    if(wv_seq[0] == 0 or wv_seq[0] == 3):
      if(a9_wv_weldingon==True):
        program_weld_on = False
        if(isHicomm):
          write_port_register(202,0)
          write_port_register(149,0)
        else:
          set_standard_digital_out(0,False)
        end
        if(wv_weldpar[2]==1):
          target_pos = feature_offset(get_actual_tcp_pose(),p[0,0,-0.01,0,0,0],wv_Line_Feature2)
          movel(target_pos,0.5,0.01)
        end
      end
    end
    background_pose = [dumy_p,dumy_p,dumy_p]
    move_p = background_pose
    return sin_dir
  end
  $ 150 "Reset"
  $ 151 "If Reset_Trig"
  if (Reset_Trig):
    $ 152 "Reset_Trig≔ False "
    global Reset_Trig=  False
    $ 153 "Call robotand_cell_initalizat"
    robotand_cell_initalizat()
    $ 154 "Auto_trig≔ False "
    global Auto_trig=  False
    $ 155 "write_port_register(cell_3f_2f_151,0)"
    write_port_register(cell_3f_2f_151,0)
    $ 156 "write_port_register(cell_info_152,0)"
    write_port_register(cell_info_152,0)
    $ 157 "write_port_register(weld_req_153,0)"
    write_port_register(weld_req_153,0)
    $ 158 "write_port_register(return_done_240,0)"
    write_port_register(return_done_240,0)
    $ 159 "write_port_register(robot_move_163,0)"
    write_port_register(robot_move_163,0)
    $ 160 "write_port_register(robot_pose_164,0)"
    write_port_register(robot_pose_164,0)
    $ 161 "write_port_register(182,0)"
    write_port_register(182,0)
    $ 162 "write_port_register(185,0)"
    write_port_register(185,0)
    $ 163 "write_port_register(201,0)"
    write_port_register(201,0)
    $ 164 "write_port_register(202,0)"
    write_port_register(202,0)
  end
  $ 165 "Welding_Init"
  $ 166 "'welding parameter initialization'"
  # 'welding parameter initialization'
  $ 167 "welding_etc"
  $ 195 "c5_wv_gap_y≔0"
  global c5_wv_gap_y=0
  $ 196 "c6_wv_gap_cpm≔0"
  global c6_wv_gap_cpm=0
  $ 197 "c9_wv_gap_freq≔0"
  global c9_wv_gap_freq=0
  $ 198 "c4_gap_enable≔0"
  global c4_gap_enable=0
  $ 199 "c7_wv_gap≔[c4_gap_enable,c5_wv_gap_y,c6_wv_gap_cpm,c9_wv_gap_freq]"
  global c7_wv_gap=[c4_gap_enable,c5_wv_gap_y,c6_wv_gap_cpm,c9_wv_gap_freq]
  $ 200 "init_reset_modbus_server"
  $ 201 "set_tool_voltage(24)"
  set_tool_voltage(24)
  $ 202 "write_port_register(163,0)"
  write_port_register(163,0)
  $ 203 "write_port_register(164,0)"
  write_port_register(164,0)
  $ 205 "write_port_register(201,1)"
  write_port_register(201,1)
  $ 206 "write_port_register(202,0)"
  write_port_register(202,0)
  $ 1235 "Thread_2"
  thread Thread_2():
    while (True):
      $ 1236 "heartbeat≔heartbeat+1"
      global heartbeat=heartbeat+1
      $ 1237 "If heartbeat>499"
      if (heartbeat>499):
        $ 1238 "heartbeat≔0"
        global heartbeat=0
      end
      $ 1239 "write_port_register(128,heartbeat)"
      write_port_register(128,heartbeat)
      $ 1249 "Wait: 1.0"
      sleep(1.0)
    end
  end
  threadId_Thread_2 = run Thread_2()
  $ 1250 "Thread_1"
  thread Thread_1():
    while (True):
      $ 1251 "a0_Job_Mode≔read_port_register(162)"
      global a0_Job_Mode= read_port_register (162)
      $ 1252 "a1_job_move≔read_port_register(163)"
      global a1_job_move= read_port_register (163)
      $ 1253 "If red_led≟ True "
      if (get_tool_digital_out(0) ==   True  ):
        $ 1254 "Set red_led=Off"
        set_tool_digital_out(0, False)
      end
      $ 1255 "If a0_Job_Mode≟2"
      if (a0_Job_Mode == 2):
        $ 1256 "If read_port_register(arc_onoff_168)≟2"
        if ( read_port_register (arc_onoff_168) == 2):
          $ 1257 "a9_wv_weldingon≔ True "
          global a9_wv_weldingon=  True
        else:
          $ 1258 "Else" "noBreak"
          $ 1259 "a9_wv_weldingon≔ False "
          global a9_wv_weldingon=  False
        end
        $ 1260 "If Auto_trig"
        if (Auto_trig):
          $ 1261 "get_next_number≔read_port_register(166)"
          global get_next_number= read_port_register (166)
          $ 1262 "get_move_trig≔read_port_register(167)"
          global get_move_trig= read_port_register (167)
          $ 1263 "If get_move_trig≟1 and running_trig≟ True "
          if (get_move_trig == 1  and  running_trig ==   True  ):
            $ 1264 "If get_next_number<0 or get_next_number>30"
            if (get_next_number<0  or  get_next_number>30):
              $ 1265 "write_port_register(142,141)"
              write_port_register(142,141)
              $ 1266 "Halt"
              halt
            end
            $ 1267 "If get_next_number≠Auto_cur_cell"
            if (get_next_number != Auto_cur_cell):
              $ 1268 "running_trig≔ False "
              global running_trig=  False
              $ 1269 "write_welder(0, False )"
              write_welder(0,  False  )
              $ 1270 "write_port_register(149,0)"
              write_port_register(149,0)
              $ 1271 "write_port_register(202,0)"
              write_port_register(202,0)
            else:
              $ 1272 "Else" "noBreak"
              $ 1273 "write_port_register(166,0)"
              write_port_register(166,0)
              $ 1274 "write_port_register(167,0)"
              write_port_register(167,0)
            end
          end
        end
        $ 1275 "If t_time>timer_1"
        if (t_time>timer_1):
          $ 1276 "write_port_register(143,timer_1)"
          write_port_register(143,timer_1)
        else:
          $ 1277 "Else" "noBreak"
          $ 1278 "write_port_register(143,timer_1)"
          write_port_register(143,timer_1)
          $ 1279 "write_port_register(144,timer_1)"
          write_port_register(144,timer_1)
        end
        $ 1280 "Monitoring touch and welding"
        $ 1281 "If read_welder_control(0) and read_port_register(130)≠1"
        if (read_welder_control(0)  and   read_port_register (130) != 1):
          $ 1282 "write_port_register(130,1)"
          write_port_register(130,1)
        else:
          $ 1283 "ElseIf read_welder_control(0) and read_port_register(130)≠0"
          if (read_welder_control(0)  and   read_port_register (130) != 0):
            $ 1284 "write_port_register(130,0)"
            write_port_register(130,0)
          end
        end
        $ 1285 "If read_welder(5)"
        if (read_welder(5)):
          $ 1286 "'check wcr in (digital)'"
          # 'check wcr in (digital)'
          $ 1287 "write_output_float_register(20,1)"
          write_output_float_register(20,1)
        else:
          $ 1288 "Else" "noBreak"
          $ 1289 "write_output_float_register(20,0)"
          write_output_float_register(20,0)
        end
        $ 1290 "If read_welder(4)"
        if (read_welder(4)):
          $ 1291 "'check touch (digital)'"
          # 'check touch (digital)'
          $ 1292 "write_output_float_register(21,1)"
          write_output_float_register(21,1)
        else:
          $ 1293 "Else" "noBreak"
          $ 1294 "write_output_float_register(21,0)"
          write_output_float_register(21,0)
        end
        $ 1295 "If read_welder_control(0)"
        if (read_welder_control(0)):
          $ 1296 "'check welding out (digital)'"
          # 'check welding out (digital)'
          $ 1297 "write_output_float_register(17,1)"
          write_output_float_register(17,1)
        else:
          $ 1298 "Else" "noBreak"
          $ 1299 "write_output_float_register(17,0)"
          write_output_float_register(17,0)
        end
        $ 1300 "If read_welder_control(4)"
        if (read_welder_control(4)):
          $ 1301 "'check touch out (digital)'"
          # 'check touch out (digital)'
          $ 1302 "write_output_float_register(18,1)"
          write_output_float_register(18,1)
        else:
          $ 1303 "Else" "noBreak"
          $ 1304 "write_output_float_register(18,0)"
          write_output_float_register(18,0)
        end
      end
      $ 1305 "If get_tool_digital_in(1)≟ True "
      if (get_tool_digital_in(1) ==   True  ):
        $ 1306 "set_tool_digital_out(1, False )"
        set_tool_digital_out(1,  False  )
      else:
        $ 1307 "Else" "noBreak"
        $ 1308 "set_tool_digital_out(1, True )"
        set_tool_digital_out(1,  True  )
      end
      $ 1309 "If red_led≟ True "
      if (get_tool_digital_out(0) ==   True  ):
        $ 1310 "Set red_led=Off"
        set_tool_digital_out(0, False)
        $ 1311 "end_freedrive_mode()"
        end_freedrive_mode()
      end
      $ 1312 "check_speed()"
      check_speed()
      $ 1313 "Wait: 0.05"
      sleep(0.05)
    end
  end
  threadId_Thread_1 = run Thread_1()
  thread EventThread():
    while (True):
      if (event_cal_on):
        $ 1317 "move_i_f≔1"
        global move_i_f=1
        $ 1318 "get_pose_side≔0"
        global get_pose_side=0
        $ 1319 "Loop move_i_f<10"
        while (move_i_f<10):
          $ 1320 "If A_Touch_trig_l[move_i_f]≟ True "
          if (A_Touch_trig_l[move_i_f] ==   True  ):
            $ 1321 "If move_i_f≟A_VL1 or move_i_f≟A_VL2"
            if (move_i_f == A_VL1  or  move_i_f == A_VL2):
              $ 1322 "A_sel_v≔move_i_f"
              global A_sel_v=move_i_f
              $ 1323 "If simulation_mode"
              if (simulation_mode):
                $ 1324 "Call welding_parameter_sim"
                welding_parameter_sim()
              else:
                $ 1325 "Else" "noBreak"
                $ 1326 "Call welding_parameter_init"
                welding_parameter_init()
              end
              $ 1327 "If a8_wv_distance<5"
              if (a8_wv_distance<5):
                $ 1328 "write_port_register(142,143)"
                write_port_register(142,143)
                $ 1329 "Halt"
                halt
              end
              $ 1330 "b2_left_par≔ True "
              global b2_left_par=  True
              $ 1331 "b8_wv_2f≔ False "
              global b8_wv_2f=  False
              $ 1332 "If move_i_f≟A_VL2"
              if (move_i_f == A_VL2):
                $ 1333 "callar_hor≔a6_callar_hor"
                global callar_hor=a6_callar_hor
                $ 1334 "b2_cell≔0"
                global b2_cell=0
                $ 1335 "If b1_cell_info_L≟c or b1_cell_info_L≟d"
                if (b1_cell_info_L == c  or  b1_cell_info_L == d):
                  $ 1336 "b2_cell≔b1_cell_info_L"
                  global b2_cell=b1_cell_info_L
                else:
                  $ 1337 "Else" "noBreak"
                  $ 1338 "b2_cell≔0"
                  global b2_cell=0
                end
              else:
                $ 1339 "Else" "noBreak"
                $ 1340 "callar_hor≔0"
                global callar_hor=0
                $ 1341 "b2_cell≔b1_cell_info_L"
                global b2_cell=b1_cell_info_L
              end
              $ 1342 "get_pos≔get_lr(left,a6_f_width,a5_f_hole,a7_f_distance,b2_left_par,b8_wv_2f,Touch_dis,get_margin_z,get_pose_side,callar_hor,b2_cell,center_line)"
              global get_pos=get_lr(p[.480496318984, .411279115151, .006998291210, -2.211681476386, -.899147924387, -1.383032568605],a6_f_width,a5_f_hole,a7_f_distance,b2_left_par,b8_wv_2f,Touch_dis,get_margin_z,get_pose_side,callar_hor,b2_cell,center_line)
              $ 1343 "pre_tp≔tilt_3f_fun(get_pos,[0,0,0],0)"
              global pre_tp=tilt_3f_fun(get_pos,[0,0,0],0)
              $ 1344 "A_Prepos_l[move_i_f]=pre_tp"
              A_Prepos_l[move_i_f]=pre_tp
            else:
              $ 1345 "ElseIf move_i_f≟A_VR1 or move_i_f≟A_VR2"
              if (move_i_f == A_VR1  or  move_i_f == A_VR2):
                $ 1346 "A_sel_v≔move_i_f"
                global A_sel_v=move_i_f
                $ 1347 "If simulation_mode"
                if (simulation_mode):
                  $ 1348 "Call welding_parameter_sim"
                  welding_parameter_sim()
                else:
                  $ 1349 "Else" "noBreak"
                  $ 1350 "Call welding_parameter_init"
                  welding_parameter_init()
                end
                $ 1351 "If a8_wv_distance<5"
                if (a8_wv_distance<5):
                  $ 1352 "write_port_register(142,143)"
                  write_port_register(142,143)
                  $ 1353 "Halt"
                  halt
                end
                $ 1354 "b2_left_par≔ False "
                global b2_left_par=  False
                $ 1355 "b8_wv_2f≔ False "
                global b8_wv_2f=  False
                $ 1356 "If move_i_f≟A_VR2"
                if (move_i_f == A_VR2):
                  $ 1357 "callar_hor≔a6_callar_hor"
                  global callar_hor=a6_callar_hor
                  $ 1358 "If b1_cell_info_R≟c or b1_cell_info_R≟d"
                  if (b1_cell_info_R == c  or  b1_cell_info_R == d):
                    $ 1359 "b2_cell≔b1_cell_info_R"
                    global b2_cell=b1_cell_info_R
                  else:
                    $ 1360 "Else" "noBreak"
                    $ 1361 "b2_cell≔0"
                    global b2_cell=0
                  end
                else:
                  $ 1362 "Else" "noBreak"
                  $ 1363 "callar_hor≔0"
                  global callar_hor=0
                  $ 1364 "b2_cell≔b1_cell_info_R"
                  global b2_cell=b1_cell_info_R
                end
                $ 1365 "get_pos≔get_lr(right,a6_f_width,a5_f_hole,a7_f_distance,b2_left_par,b8_wv_2f,Touch_dis,get_margin_z,get_pose_side,callar_hor,b2_cell,center_line)"
                global get_pos=get_lr(p[.475000000000, -.421403215678, .026417194146, 1.917761036827, -1.141682393512, 1.523356199292],a6_f_width,a5_f_hole,a7_f_distance,b2_left_par,b8_wv_2f,Touch_dis,get_margin_z,get_pose_side,callar_hor,b2_cell,center_line)
                $ 1366 "pre_tp≔tilt_3f_fun(get_pos,[0,0,0],0)"
                global pre_tp=tilt_3f_fun(get_pos,[0,0,0],0)
                $ 1367 "A_Prepos_l[move_i_f]=pre_tp"
                A_Prepos_l[move_i_f]=pre_tp
              else:
                $ 1368 "ElseIf move_i_f≟A_HOR"
                if (move_i_f == A_HOR):
                  $ 1369 "A_sel_v≔A_HOR"
                  global A_sel_v=A_HOR
                  $ 1370 "If simulation_mode"
                  if (simulation_mode):
                    $ 1371 "Call welding_parameter_sim"
                    welding_parameter_sim()
                  else:
                    $ 1372 "Else" "noBreak"
                    $ 1373 "Call welding_parameter_init"
                    welding_parameter_init()
                  end
                  $ 1374 "b8_wv_2f≔ True "
                  global b8_wv_2f=  True
                  $ 1375 "b2_left_par≔ True "
                  global b2_left_par=  True
                  $ 1376 "b2_cell≔b1_cell_info_L"
                  global b2_cell=b1_cell_info_L
                  $ 1377 "get_pos≔get_lr(up_left,a6_f_width,a5_f_hole,a7_f_distance,b2_left_par,b8_wv_2f,Touch_dis,get_margin_z,get_pose_side,0,b2_cell,center_line)"
                  global get_pos=get_lr(p[.492775857339, .409517380626, -.029063830209, -2.419264859926, -.998084331190, -1.368689080860],a6_f_width,a5_f_hole,a7_f_distance,b2_left_par,b8_wv_2f,Touch_dis,get_margin_z,get_pose_side,0,b2_cell,center_line)
                  $ 1378 "pre_tp≔get_pos"
                  global pre_tp=get_pos
                  $ 1379 "A_Prepos_l[move_i_f]=pre_tp"
                  A_Prepos_l[move_i_f]=pre_tp
                else:
                  $ 1380 "ElseIf move_i_f≟A_HOR_R"
                  if (move_i_f == A_HOR_R):
                    $ 1381 "A_sel_v≔A_HOR"
                    global A_sel_v=A_HOR
                    $ 1382 "If simulation_mode"
                    if (simulation_mode):
                      $ 1383 "Call welding_parameter_sim"
                      welding_parameter_sim()
                    else:
                      $ 1384 "Else" "noBreak"
                      $ 1385 "Call welding_parameter_init"
                      welding_parameter_init()
                    end
                    $ 1386 "b2_left_par≔ False "
                    global b2_left_par=  False
                    $ 1387 "b8_wv_2f≔ True "
                    global b8_wv_2f=  True
                    $ 1388 "b2_cell≔b1_cell_info_R"
                    global b2_cell=b1_cell_info_R
                    $ 1389 "get_pos≔get_lr(up_right,a6_f_width,a5_f_hole,a7_f_distance,b2_left_par,b8_wv_2f,Touch_dis,get_margin_z,get_pose_side,0,b2_cell,center_line)"
                    global get_pos=get_lr(p[.445203173045, -.406687378356, -.031125942276, 2.308490741423, -1.066468937023, 1.322151316133],a6_f_width,a5_f_hole,a7_f_distance,b2_left_par,b8_wv_2f,Touch_dis,get_margin_z,get_pose_side,0,b2_cell,center_line)
                    $ 1390 "pre_tp≔get_pos"
                    global pre_tp=get_pos
                    $ 1391 "A_Prepos_l[move_i_f]=pre_tp"
                    A_Prepos_l[move_i_f]=pre_tp
                  else:
                    $ 1392 "ElseIf move_i_f≟A_HOR_ML"
                    if (move_i_f == A_HOR_ML):
                      $ 1393 "A_sel_v≔A_HOR_ML"
                      global A_sel_v=A_HOR_ML
                      $ 1394 "If simulation_mode"
                      if (simulation_mode):
                        $ 1395 "Call welding_parameter_sim"
                        welding_parameter_sim()
                      else:
                        $ 1396 "Else" "noBreak"
                        $ 1397 "Call welding_parameter_init"
                        welding_parameter_init()
                      end
                      $ 1398 "b8_wv_2f≔ True "
                      global b8_wv_2f=  True
                      $ 1399 "b2_left_par≔ True "
                      global b2_left_par=  True
                      $ 1400 "b2_cell≔b1_cell_info_L"
                      global b2_cell=b1_cell_info_L
                      $ 1401 "Touch_dis≔-1*Touch_dis"
                      global Touch_dis=-1*Touch_dis
                      $ 1402 "get_pos≔get_lr(up_left,a6_f_width,a5_f_hole,a7_f_distance,b2_left_par,b8_wv_2f,Touch_dis,get_margin_z,get_pose_side,a6_callar_hor,b2_cell,center_line)"
                      global get_pos=get_lr(p[.492775857339, .409517380626, -.029063830209, -2.419264859926, -.998084331190, -1.368689080860],a6_f_width,a5_f_hole,a7_f_distance,b2_left_par,b8_wv_2f,Touch_dis,get_margin_z,get_pose_side,a6_callar_hor,b2_cell,center_line)
                      $ 1403 "Touch_dis≔-1*Touch_dis"
                      global Touch_dis=-1*Touch_dis
                      $ 1404 "pre_tp≔get_pos"
                      global pre_tp=get_pos
                      $ 1405 "A_Prepos_l[move_i_f]=pre_tp"
                      A_Prepos_l[move_i_f]=pre_tp
                    else:
                      $ 1406 "ElseIf move_i_f≟A_HOR_MR"
                      if (move_i_f == A_HOR_MR):
                        $ 1407 "A_sel_v≔A_HOR_MR"
                        global A_sel_v=A_HOR_MR
                        $ 1408 "If simulation_mode"
                        if (simulation_mode):
                          $ 1409 "Call welding_parameter_sim"
                          welding_parameter_sim()
                        else:
                          $ 1410 "Else" "noBreak"
                          $ 1411 "Call welding_parameter_init"
                          welding_parameter_init()
                        end
                        $ 1412 "b2_left_par≔ False "
                        global b2_left_par=  False
                        $ 1413 "b8_wv_2f≔ True "
                        global b8_wv_2f=  True
                        $ 1414 "b2_cell≔b1_cell_info_R"
                        global b2_cell=b1_cell_info_R
                        $ 1415 "Touch_dis≔-1*Touch_dis"
                        global Touch_dis=-1*Touch_dis
                        $ 1416 "get_pos≔get_lr(up_right,a6_f_width,a5_f_hole,a7_f_distance,b2_left_par,b8_wv_2f,Touch_dis,get_margin_z,get_pose_side,a6_callar_hor,b2_cell,center_line)"
                        global get_pos=get_lr(p[.445203173045, -.406687378356, -.031125942276, 2.308490741423, -1.066468937023, 1.322151316133],a6_f_width,a5_f_hole,a7_f_distance,b2_left_par,b8_wv_2f,Touch_dis,get_margin_z,get_pose_side,a6_callar_hor,b2_cell,center_line)
                        $ 1417 "Touch_dis≔-1*Touch_dis"
                        global Touch_dis=-1*Touch_dis
                        $ 1418 "pre_tp≔get_pos"
                        global pre_tp=get_pos
                        $ 1419 "A_Prepos_l[move_i_f]=pre_tp"
                        A_Prepos_l[move_i_f]=pre_tp
                      end
                    end
                  end
                end
              end
            end
            $ 1420 "If move_i_f≤4"
            if (move_i_f <= 4):
              $ 1421 "A_Prepos_l[move_i_f+9]=p[0,0,0,0,0,0]"
              A_Prepos_l[move_i_f+9]=p[0,0,0,0,0,0]
            end
          end
          $ 1424 "move_i_f≔move_i_f+1"
          global move_i_f=move_i_f+1
        end
        $ 1425 "event_cal_on≔ False "
        global event_cal_on=  False
      elif (event_side_on):
        $ 1429 "Wait event_cal_on≟ False "
        while (not(event_cal_on ==   False  )):
          sync()
        end
        $ 1430 "move_i_f≔1"
        global move_i_f=1
        $ 1431 "get_pose_side≔get_pose_side_t"
        global get_pose_side=get_pose_side_t
        $ 1432 "Loop move_i_f<10"
        while (move_i_f<10):
          $ 1433 "If A_Touch_trig_l[move_i_f]≟ True "
          if (A_Touch_trig_l[move_i_f] ==   True  ):
            $ 1434 "If move_i_f≟A_VL1 or move_i_f≟A_VL2"
            if (move_i_f == A_VL1  or  move_i_f == A_VL2):
              $ 1435 "A_Prepos_l[move_i_f]=side_apply(A_Prepos_l[move_i_f],center_line,get_pose_side)"
              A_Prepos_l[move_i_f]=side_apply(A_Prepos_l[move_i_f],center_line,get_pose_side)
            else:
              $ 1436 "ElseIf move_i_f≟A_VR1 or move_i_f≟A_VR2"
              if (move_i_f == A_VR1  or  move_i_f == A_VR2):
                $ 1437 "A_Prepos_l[move_i_f]=side_apply(A_Prepos_l[move_i_f],center_line,get_pose_side)"
                A_Prepos_l[move_i_f]=side_apply(A_Prepos_l[move_i_f],center_line,get_pose_side)
              else:
                $ 1438 "ElseIf move_i_f≟A_HOR"
                if (move_i_f == A_HOR):
                  $ 1439 "A_Prepos_l[move_i_f]=side_apply(A_Prepos_l[move_i_f],center_line,get_pose_side)"
                  A_Prepos_l[move_i_f]=side_apply(A_Prepos_l[move_i_f],center_line,get_pose_side)
                else:
                  $ 1440 "ElseIf move_i_f≟A_HOR_R"
                  if (move_i_f == A_HOR_R):
                    $ 1441 "A_Prepos_l[move_i_f]=side_apply(A_Prepos_l[move_i_f],center_line,get_pose_side)"
                    A_Prepos_l[move_i_f]=side_apply(A_Prepos_l[move_i_f],center_line,get_pose_side)
                  else:
                    $ 1442 "ElseIf move_i_f≟A_HOR_ML"
                    if (move_i_f == A_HOR_ML):
                      $ 1443 "A_Prepos_l[move_i_f]=side_apply(A_Prepos_l[move_i_f],center_line,get_pose_side)"
                      A_Prepos_l[move_i_f]=side_apply(A_Prepos_l[move_i_f],center_line,get_pose_side)
                    else:
                      $ 1444 "ElseIf move_i_f≟A_HOR_MR"
                      if (move_i_f == A_HOR_MR):
                        $ 1445 "A_Prepos_l[move_i_f]=side_apply(A_Prepos_l[move_i_f],center_line,get_pose_side)"
                        A_Prepos_l[move_i_f]=side_apply(A_Prepos_l[move_i_f],center_line,get_pose_side)
                      end
                    end
                  end
                end
              end
            end
          end
          $ 1446 "move_i_f≔move_i_f+1"
          global move_i_f=move_i_f+1
        end
        $ 1447 "event_side_on≔ False "
        global event_side_on=  False
      elif (reset_trig):
        $ 1449 "Call reset_weld_param"
        reset_weld_param()
        $ 1450 "reset_trig≔ False "
        global reset_trig=  False
      elif (time_cal_trig):
        $ 1452 "t_time≔time_cal(Auto_W_num,Auto_total_cell,A_Speed_list,A_Distance_list,A_Touch_p,0)"
        global t_time=time_cal(Auto_W_num,Auto_total_cell,A_Speed_list,A_Distance_list,A_Touch_p,0)
        $ 1453 "write_port_register(144,t_time)"
        write_port_register(144,t_time)
        $ 1454 "time_cal_trig≔ False "
        global time_cal_trig=  False
      elif (pause_trig):
        $ 1456 "s_conn≔socket_open('192.168.1.7',29999)"
        global s_conn=socket_open("192.168.1.7",29999)
        $ 1457 "s_send≔socket_send_string('pause')"
        global s_send=socket_send_string("pause")
        $ 1458 "s_send≔socket_send_byte(10)"
        global s_send=socket_send_byte(10)
        $ 1459 "socket_close()"
        socket_close()
        $ 1460 "pause_trig≔ False "
        global pause_trig=  False
      end
      sync()
    end
  end
  eventThread = run EventThread()
  while (True):
    $ 207 "Robot Program"
    $ 225 "If simulation_mode"
    if (simulation_mode):
      $ 226 "'work mode 2'"
      # 'work mode 2'
      $ 227 "write_port_register(162,2)"
      write_port_register(162,2)
      $ 228 "touch_temp≔0"
      global touch_temp=0
    end
    $ 229 "If a0_Job_Mode≟1"
    if (a0_Job_Mode == 1):
      $ 230 "job mode 1"
      $ 231 "'JOB_MANUAL'"
      # 'JOB_MANUAL'
      $ 232 "write_port_register(robot_ready_141,1)"
      write_port_register(robot_ready_141,1)
      $ 233 "If freedrive≟ True  and freedrive_trg≟ False "
      if (get_tool_digital_in(1) ==   True    and  freedrive_trg ==   False  ):
        $ 234 "freedrive_trg≔ True "
        global freedrive_trg=  True
        $ 235 "freedrive_mode()"
        freedrive_mode()
      else:
        $ 236 "ElseIf freedrive≟ False  and freedrive_trg≟ True "
        if (get_tool_digital_in(1) ==   False    and  freedrive_trg ==   True  ):
          $ 237 "end_freedrive_mode()"
          end_freedrive_mode()
          $ 238 "freedrive_trg≔ False "
          global freedrive_trg=  False
        end
      end
      $ 242 "If freedrive≟ True  and save_tool≟ True "
      if (get_tool_digital_in(1) ==   True    and  get_tool_digital_in(0) ==   True  ):
        $ 246 "Wait: 0.01"
        sleep(0.01)
      else:
        $ 247 "ElseIf a1_job_move≟1"
        if (a1_job_move == 1):
          $ 248 "'Manual - Move Home/Packing/Warmup'"
          # 'Manual - Move Home/Packing/Warmup'
          $ 249 "If read_port_register(robot_pose_164)≟1"
          if ( read_port_register (robot_pose_164) == 1):
            $ 250 "write_port_register(robot_ready_141,0)"
            write_port_register(robot_ready_141,0)
            $ 251 "homeing()"
            homeing()
            $ 252 "MoveJ"
            $ 253 "Packing_pos" "breakAfter"
            movej([1.5877798795700073, -0.0173419157611292, -2.4983108679400843, -1.4065726439105433, 1.626846194267273, 3.0169763565063477], a=0.9599310885968813, v=0.9599310885968813)
          else:
            $ 254 "ElseIf read_port_register(robot_pose_164)≟2"
            if ( read_port_register (robot_pose_164) == 2):
              $ 255 "write_port_register(robot_ready_141,0)"
              write_port_register(robot_ready_141,0)
              $ 256 "homeing()"
              homeing()
            else:
              $ 257 "ElseIf read_port_register(robot_pose_164)≟3"
              global thread_flag_257=0
              thread Thread_if_257():
                $ 258 "write_port_register(robot_ready_141,0)"
                write_port_register(robot_ready_141,0)
                $ 259 "Warm-up"
                $ 260 "Loop 22 times"
                Loop_9 = 0
                while (Loop_9 < 22):
                  $ 261 "MoveJ"
                  $ 262 "Warming_1" "breakAfter"
                  movej([1.3388409470167426, -1.0894445773085817, -1.21578769245379, -2.340308120379028, 1.4975742894997062, 2.3546781160711117], a=0.5235987755982988, v=0.2617993877991494)
                  $ 263 "Warming_2" "breakAfter"
                  movej([0.3765170846483107, -1.0894466320678031, -1.215768207322279, -2.3402268007341895, 1.4977834941028334, 2.3545507363355367], a=0.5235987755982988, v=0.2617993877991494)
                  $ 264 "Warming_3" "breakAfter"
                  movej([0.70229908534082, -1.0894474234917375, -1.2158576930717002, -2.340314378048955, 1.497725846219038, 2.3545705560997385], a=0.5235987755982988, v=0.2617993877991494)
                  $ 265 "Warming_4" "breakAfter"
                  movej([0.7262700130956564, -1.3120291852612347, -1.2099656497338014, -2.3525900953229293, 1.4887798341942113, 2.3787312683819053], a=0.5235987755982988, v=0.2617993877991494)
                  $ 266 "Wariming_5" "breakAfter"
                  movej([0.6926726182060315, -1.0476106481659855, -1.2179788018883642, -2.3355421428203886, 1.501172277634622, 2.3452576869092923], a=0.5235987755982988, v=0.2617993877991494)
                  $ 267 "Warming_6" "breakAfter"
                  movej([0.706544616734295, -1.047040496424307, -1.4190888321133315, -2.3436933501169452, 1.4896422361111494, 2.359727124413684], a=0.5235987755982988, v=0.2617993877991494)
                  $ 268 "Warming_7" "breakAfter"
                  movej([0.6929880468286825, -1.0476354157293724, -1.2203987593812862, -2.335678707355349, 1.5010671072282735, 2.34550338764565], a=0.5235987755982988, v=0.2617993877991494)
                  $ 269 "Warming_8" "breakAfter"
                  movej([0.6920775233962951, -1.0506328608604214, -1.2152130579572011, -2.5072867131215766, 1.4917910996963177, 2.3459413556024855], a=0.5235987755982988, v=0.2617993877991494)
                  $ 270 "Warming_9" "breakAfter"
                  movej([0.692933302781529, -1.0474869681006531, -1.2206503884398048, -2.327559666709858, 1.5015191668476027, 2.3454614641680087], a=0.5235987755982988, v=0.2617993877991494)
                  $ 271 "Warming_10" "breakAfter"
                  movej([0.7189566793816887, -1.1462083943843844, -1.3286482352122917, -2.3898368690561114, 1.223390234561962, 2.3705741030878644], a=0.5235987755982988, v=0.2617993877991494)
                  $ 272 "Warming_11" "breakAfter"
                  movej([0.6952417412291937, -1.0226626805382075, -1.3187663864026051, -2.3852732107244847, 1.5281305955128988, 2.3484138521676003], a=0.5235987755982988, v=0.2617993877991494)
                  $ 273 "Warming_12" "breakAfter"
                  movej([0.6939658935868351, -1.0222541193887693, -1.3205060700309819, -2.4036431483224994, 1.8876292979334401, 2.3447872177861786], a=0.5235987755982988, v=0.2617993877991494)
                  $ 274 "Warming_13" "breakAfter"
                  movej([0.6855475262233561, -1.0389108716421376, -1.3163550590643318, -2.371185255756596, 1.5282046997566647, 1.6427118007650936], a=0.5235987755982988, v=0.2617993877991494)
                  $ 275 "Warming_14" "breakAfter"
                  movej([0.721349856763205, -1.0075982028648234, -1.3205933019427434, -2.399656340024448, 1.5281938267886401, 2.9170078642332813], a=0.5235987755982988, v=0.2617993877991494)
                  Loop_9 = Loop_9 + 1
                end
                $ 276 "homeing()"
                homeing()
                $ 277 "Wait: 2.0"
                sleep(2.0)
                thread_flag_257 = 1
              end
              if ( read_port_register (robot_pose_164) == 3):
                global thread_handler_257=run Thread_if_257()
                while (thread_flag_257 == 0):
                  if not( read_port_register (robot_pose_164) == 3):
                    kill thread_handler_257
                    thread_flag_257 = 2
                  else:
                    sync()
                  end
                end
              else:
                thread_flag_257 = 2
              end
              if (thread_flag_257 == 2):
                $ 278 "ElseIf read_port_register(robot_pose_164)≟4"
                if ( read_port_register (robot_pose_164) == 4):
                  $ 279 "write_port_register(robot_ready_141,0)"
                  write_port_register(robot_ready_141,0)
                  $ 280 "homeing()"
                  homeing()
                  $ 281 "MoveJ"
                  $ 282 "pre_mounting" "breakAfter"
                  movej([1.2356762886047363, -0.8703244368182581, -0.942230526600973, -2.3905327955829065, 1.3216267824172974, 2.6514604091644287], a=0.7853981633974483, v=0.7853981633974483)
                  $ 283 "Mounting_pos" "breakAfter"
                  movej([0.6231353085164267, -0.6300961531972575, -0.9034285948871803, -1.770059340221131, 1.417516049558281, 1.7792033261567348], a=0.7853981633974483, v=0.7853981633974483)
                else:
                  $ 284 "ElseIf read_port_register(robot_pose_164)≟5"
                  if ( read_port_register (robot_pose_164) == 5):
                    $ 285 "c_p≔get_actual_tcp_pose()"
                    global c_p= get_actual_tcp_pose ()
                    $ 286 "MoveL"
                    $ 287 "m_p≔pose_trans(c_p, p[0,0,0,d2r(tilt_deg_man),0,0])"
                    global m_p= pose_trans (c_p, p[0,0,0,d2r(tilt_deg_man),0,0])
                    $ 288 "m_p" "breakAfter"
                    movel(pose_trans(Base, m_p), a=0.03, v=0.03)
                    $ 289 "m_p≔pose_trans(c_p, p[0,0,0,d2r(-tilt_deg_man),0,0])"
                    global m_p= pose_trans (c_p, p[0,0,0,d2r(-tilt_deg_man),0,0])
                    $ 290 "m_p" "breakAfter"
                    movel(pose_trans(Base, m_p), a=0.03, v=0.03)
                    $ 291 "c_p" "breakAfter"
                    movel(pose_trans(Base, c_p), a=0.03, v=0.03)
                    $ 292 "m_p≔pose_trans(c_p, p[0,0,0,0,d2r(tilt_deg_man),0])"
                    global m_p= pose_trans (c_p, p[0,0,0,0,d2r(tilt_deg_man),0])
                    $ 293 "m_p" "breakAfter"
                    movel(pose_trans(Base, m_p), a=0.03, v=0.03)
                    $ 294 "m_p≔pose_trans(c_p, p[0,0,0,0,d2r(-tilt_deg_man),0])"
                    global m_p= pose_trans (c_p, p[0,0,0,0,d2r(-tilt_deg_man),0])
                    $ 295 "m_p" "breakAfter"
                    movel(pose_trans(Base, m_p), a=0.03, v=0.03)
                    $ 296 "c_p" "breakAfter"
                    movel(pose_trans(Base, c_p), a=0.03, v=0.03)
                    $ 297 "m_p≔pose_trans(c_p, p[0,0,0,0,0,d2r(tilt_deg_man)])"
                    global m_p= pose_trans (c_p, p[0,0,0,0,0,d2r(tilt_deg_man)])
                    $ 298 "m_p" "breakAfter"
                    movel(pose_trans(Base, m_p), a=0.03, v=0.03)
                    $ 299 "m_p≔pose_trans(c_p, p[0,0,0,0,0,d2r(-tilt_deg_man)])"
                    global m_p= pose_trans (c_p, p[0,0,0,0,0,d2r(-tilt_deg_man)])
                    $ 300 "m_p" "breakAfter"
                    movel(pose_trans(Base, m_p), a=0.03, v=0.03)
                    $ 301 "c_p" "breakAfter"
                    movel(pose_trans(Base, c_p), a=0.03, v=0.03)
                  end
                end
              end
            end
          end
          $ 302 "Call Move_done"
          Move_done()
        end
      end
      $ 303 "Call robotand_cell_initalizat"
      robotand_cell_initalizat()
    else:
      $ 304 "ElseIf a0_Job_Mode≟2"
      global thread_flag_304=0
      thread Thread_if_304():
        $ 305 "'JOB_AUTO'"
        # 'JOB_AUTO'
        $ 306 "auto_on≔ True "
        global auto_on=  True
        $ 307 "Init"
        $ 308 "If freedrive_trg"
        if (freedrive_trg):
          $ 309 "end_freedrive_mode()"
          end_freedrive_mode()
          $ 310 "freedrive_trg≔ False "
          global freedrive_trg=  False
        end
        $ 311 "write_port_register(202,0)"
        write_port_register(202,0)
        $ 312 "write_port_register(robot_ready_141,0)"
        write_port_register(robot_ready_141,0)
        $ 313 "homeing()"
        homeing()
        $ 314 "Wait: 0.2"
        sleep(0.2)
        $ 315 "Cell_calculation"
        $ 316 "'setting'"
        # 'setting'
        $ 317 "Auto_trig≔ False "
        global Auto_trig=  False
        $ 318 "If Auto_trig≟ False "
        if (Auto_trig ==   False  ):
          $ 319 "If simulation_mode"
          if (simulation_mode):
            $ 320 "b1_cell_info_L≔B"
            global b1_cell_info_L=B
            $ 321 "b1_cell_info_R≔B"
            global b1_cell_info_R=B
            $ 322 "b1_cell_select≔motion_num([A_VL1,A_VR1,A_HOR,0,0,0])"
            global b1_cell_select=motion_num([A_VL1,A_VR1,A_HOR,0,0,0])
            $ 323 "b1_cell_select≔motion_num([A_HOR,0,0,0,0,0])"
            global b1_cell_select=motion_num([A_HOR,0,0,0,0,0])
            $ 324 "EXT_flag1≔integer_to_binary_list(read_port_register(2048))"
            global EXT_flag1= integer_to_binary_list ( read_port_register (2048))
            $ 325 "b1_cell_thickne≔6"
            global b1_cell_thickne=6
            $ 326 "A_Touch_trig_l≔touch_cal(b1_cell_info_L,b1_cell_info_R,b1_cell_select)"
            global A_Touch_trig_l=touch_cal(b1_cell_info_L,b1_cell_info_R,b1_cell_select)
            $ 327 "Auto_W_num≔cell_motion(A_Touch_trig_l,b1_cell_thickne,EXT_flag1,b1_cell_info_L,b1_cell_info_R)"
            global Auto_W_num=cell_motion(A_Touch_trig_l,b1_cell_thickne,EXT_flag1,b1_cell_info_L,b1_cell_info_R)
            $ 329 "Auto_total_cell≔cell_num(Auto_W_num)"
            global Auto_total_cell=cell_num(Auto_W_num)
            $ 330 "Auto_trig≔ True "
            global Auto_trig=  True
            $ 331 "A_sel_v≔Auto_W_num[0]"
            global A_sel_v=Auto_W_num[0]
          else:
            $ 332 "Else" "noBreak"
            $ 333 "b1_cell_info_L≔read_port_register(171)"
            global b1_cell_info_L= read_port_register (171)
            $ 334 "b1_cell_info_R≔read_port_register(172)"
            global b1_cell_info_R= read_port_register (172)
            $ 335 "EXT_flag1≔integer_to_binary_list(read_port_register(179))"
            global EXT_flag1= integer_to_binary_list ( read_port_register (179))
            $ 336 "b1_cell_select≔read_port_register(178)"
            global b1_cell_select= read_port_register (178)
            $ 337 "b1_cell_thickne≔read_port_register(183)"
            global b1_cell_thickne= read_port_register (183)
            $ 338 "A_Touch_trig_l≔touch_cal(b1_cell_info_L,b1_cell_info_R,b1_cell_select)"
            global A_Touch_trig_l=touch_cal(b1_cell_info_L,b1_cell_info_R,b1_cell_select)
            $ 339 "Auto_W_num≔cell_motion(A_Touch_trig_l,b1_cell_thickne,EXT_flag1,b1_cell_info_L,b1_cell_info_R)"
            global Auto_W_num=cell_motion(A_Touch_trig_l,b1_cell_thickne,EXT_flag1,b1_cell_info_L,b1_cell_info_R)
            $ 340 "Auto_total_cell≔cell_num(Auto_W_num)"
            global Auto_total_cell=cell_num(Auto_W_num)
            $ 341 "Auto_trig≔ True "
            global Auto_trig=  True
            $ 342 "A_sel_v≔Auto_W_num[0]"
            global A_sel_v=Auto_W_num[0]
          end
          $ 343 "write_port_register(139,Auto_total_cell-1)"
          write_port_register(139,Auto_total_cell-1)
        end
        $ 344 "Auto_cur_cell≔0"
        global Auto_cur_cell=0
        $ 345 "Touch,Welding"
        $ 346 "'Calculate total sequence and decide way'"
        # 'Calculate total sequence and decide way'
        $ 347 "Calculate & Move & Touch"
        $ 348 "touch_init"
        $ 349 "Call cell_info"
        cell_info()
        $ 350 "If simulation_mode"
        if (simulation_mode):
          $ 351 "Call welding_parameter_sim"
          welding_parameter_sim()
        else:
          $ 352 "Else" "noBreak"
          $ 353 "Call welding_parameter_init"
          welding_parameter_init()
          $ 354 "touch_temp≔read_port_register(180)"
          global touch_temp= read_port_register (180)
          $ 355 "A_cur_2f≔0"
          global A_cur_2f=0
          $ 356 "wv_direction≔1"
          global wv_direction=1
        end
        $ 357 "If touch_temp≟0"
        if (touch_temp == 0):
          $ 358 "reset Variable"
          $ 359 "A_Prepos_l=[p[0, 0, 0, 0, 0, 0], p[0, 0, 0, 0, 0, 0], p[0, 0, 0, 0, 0, 0],p[0, 0, 0, 0, 0, 0], p[0, 0, 0, 0, 0, 0], p[0, 0, 0, 0, 0, 0], p[0, 0, 0, 0, 0, 0], p[0, 0, 0, 0, 0, 0], p[0, 0, 0, 0, 0, 0], p[0, 0, 0, 0, 0, 0], p[0, 0, 0, 0, 0, 0],p[0, 0, 0, 0, 0, 0],p[0, 0, 0, 0, 0, 0],p[0, 0, 0, 0, 0, 0],p[0, 0, 0, 0, 0, 0],p[0,0,0,0,0,0]]"
          A_Prepos_l=[p[0, 0, 0, 0, 0, 0], p[0, 0, 0, 0, 0, 0], p[0, 0, 0, 0, 0, 0],p[0, 0, 0, 0, 0, 0], p[0, 0, 0, 0, 0, 0], p[0, 0, 0, 0, 0, 0], p[0, 0, 0, 0, 0, 0], p[0, 0, 0, 0, 0, 0], p[0, 0, 0, 0, 0, 0], p[0, 0, 0, 0, 0, 0], p[0, 0, 0, 0, 0, 0],p[0, 0, 0, 0, 0, 0],p[0, 0, 0, 0, 0, 0],p[0, 0, 0, 0, 0, 0],p[0, 0, 0, 0, 0, 0],p[0,0,0,0,0,0]]
          $ 360 "A_Touch_p=[p[0, 0, 0, 0, 0, 0], p[0, 0, 0, 0, 0, 0], p[0, 0, 0, 0, 0, 0],p[0, 0, 0, 0, 0, 0], p[0, 0, 0, 0, 0, 0], p[0, 0, 0, 0, 0, 0], p[0, 0, 0, 0, 0, 0], p[0, 0, 0, 0, 0, 0], p[0, 0, 0, 0, 0, 0], p[0, 0, 0, 0, 0, 0], p[0, 0, 0, 0, 0, 0],p[0, 0, 0, 0, 0, 0],p[0, 0, 0, 0, 0, 0],p[0, 0, 0, 0, 0, 0],p[0, 0, 0, 0, 0, 0],p[0,0,0,0,0,0]]"
          A_Touch_p=[p[0, 0, 0, 0, 0, 0], p[0, 0, 0, 0, 0, 0], p[0, 0, 0, 0, 0, 0],p[0, 0, 0, 0, 0, 0], p[0, 0, 0, 0, 0, 0], p[0, 0, 0, 0, 0, 0], p[0, 0, 0, 0, 0, 0], p[0, 0, 0, 0, 0, 0], p[0, 0, 0, 0, 0, 0], p[0, 0, 0, 0, 0, 0], p[0, 0, 0, 0, 0, 0],p[0, 0, 0, 0, 0, 0],p[0, 0, 0, 0, 0, 0],p[0, 0, 0, 0, 0, 0],p[0, 0, 0, 0, 0, 0],p[0,0,0,0,0,0]]
          $ 361 "reset_par"
          $ 362 "for_cal_rot≔p[0,0,0,0,0,0]"
          global for_cal_rot=p[0,0,0,0,0,0]
          $ 363 "for_cal_zr≔p[0,0,0,0,0,0]"
          global for_cal_zr=p[0,0,0,0,0,0]
          $ 364 "for_cal_zl≔p[0,0,0,0,0,0]"
          global for_cal_zl=p[0,0,0,0,0,0]
          $ 365 "for_cal_x_wel≔p[0,0,0,0,0,0]"
          global for_cal_x_wel=p[0,0,0,0,0,0]
          $ 366 "for_cal_xy≔p[0,0,0,0,0,0]"
          global for_cal_xy=p[0,0,0,0,0,0]
          $ 367 "for_cal_y_wel≔p[0,0,0,0,0,0]"
          global for_cal_y_wel=p[0,0,0,0,0,0]
          $ 368 "for_x_HOR≔p[0,0,0,0,0,0]"
          global for_x_HOR=p[0,0,0,0,0,0]
          $ 369 "for_x_HOR_R≔p[0,0,0,0,0,0]"
          global for_x_HOR_R=p[0,0,0,0,0,0]
          $ 370 "for_z_VL1≔p[0,0,0,0,0,0]"
          global for_z_VL1=p[0,0,0,0,0,0]
          $ 371 "for_z_VR1≔p[0,0,0,0,0,0]"
          global for_z_VR1=p[0,0,0,0,0,0]
        end
        $ 372 "write_port_register(143,0)"
        write_port_register(143,0)
        $ 373 "write_port_register(144,0)"
        write_port_register(144,0)
        $ 374 "timer_1: Reset"
        timer_1 = 0
        $ 375 "EXT_flag1≔integer_to_binary_list(read_port_register(179))"
        global EXT_flag1= integer_to_binary_list ( read_port_register (179))
        $ 377 "If touch_temp≟0"
        if (touch_temp == 0):
          $ 378 "write_port_register(138,0)"
          write_port_register(138,0)
          $ 379 "get_touch_position"
          $ 380 "get pre-positions"
          $ 381 "If read_port_register(work_type_165)≟2"
          if ( read_port_register (work_type_165) == 2):
            $ 382 "freedrive touch"
            $ 383 "move_i≔1"
            global move_i=1
            $ 384 "Loop move_i<9"
            while (move_i<9):
              $ 385 "Wait: 0.1"
              sleep(0.1)
              $ 386 "Wait save_tool=LO"
              while (get_tool_digital_in(0) == True):
                sync()
              end
              $ 387 "If A_Touch_trig_l[move_i]≟ True "
              if (A_Touch_trig_l[move_i] ==   True  ):
                $ 388 "If move_i≟A_HOR"
                if (move_i == A_HOR):
                  $ 389 "If b1_cell_info_L≟B or b1_cell_info_L≟D or b1_cell_info_L≟d or A_Prepos_l[A_VL1]≟p[0,0,0,0,0,0]"
                  if (b1_cell_info_L == B  or  b1_cell_info_L == D  or  b1_cell_info_L == d  or  A_Prepos_l[A_VL1] == p[0,0,0,0,0,0]):
                    $ 390 "write_port_register(touch_cell_155,5)"
                    write_port_register(touch_cell_155,5)
                    $ 391 "write_port_register(touch_num_156,1)"
                    write_port_register(touch_num_156,1)
                    $ 392 "Call touch_sub"
                    touch_sub()
                    $ 393 "g_cp≔get_actual_tcp_pose()"
                    global g_cp= get_actual_tcp_pose ()
                    $ 394 "If g_cp[2]<(get_margin_z+a7_cell_bottom)/1000"
                    if (g_cp[2]<(get_margin_z+a7_cell_bottom)/1000):
                      $ 395 "g_cp[2]=(get_margin_z+a7_cell_bottom)/1000"
                      g_cp[2]=(get_margin_z+a7_cell_bottom)/1000
                    end
                    $ 396 "A_Prepos_l[move_i]=g_cp"
                    A_Prepos_l[move_i]=g_cp
                  end
                else:
                  $ 397 "ElseIf move_i≟A_HOR_ML"
                  if (move_i == A_HOR_ML):
                    $ 398 "If b1_cell_info_L≟B or b1_cell_info_L≟D or b1_cell_info_L≟d or A_Prepos_l[A_VL1]≟p[0,0,0,0,0,0]"
                    if (b1_cell_info_L == B  or  b1_cell_info_L == D  or  b1_cell_info_L == d  or  A_Prepos_l[A_VL1] == p[0,0,0,0,0,0]):
                      $ 399 "write_port_register(touch_cell_155,5)"
                      write_port_register(touch_cell_155,5)
                      $ 400 "write_port_register(touch_num_156,3)"
                      write_port_register(touch_num_156,3)
                      $ 401 "Call touch_sub"
                      touch_sub()
                      $ 402 "g_cp≔get_actual_tcp_pose()"
                      global g_cp= get_actual_tcp_pose ()
                      $ 403 "If g_cp[2]<(get_margin_z+a7_cell_bottom)/1000"
                      if (g_cp[2]<(get_margin_z+a7_cell_bottom)/1000):
                        $ 404 "g_cp[2]=(get_margin_z+a7_cell_bottom)/1000"
                        g_cp[2]=(get_margin_z+a7_cell_bottom)/1000
                      end
                      $ 405 "A_Prepos_l[move_i]=g_cp"
                      A_Prepos_l[move_i]=g_cp
                    end
                  else:
                    $ 406 "ElseIf move_i≟A_HOR_R"
                    if (move_i == A_HOR_R):
                      $ 407 "If b1_cell_info_L≟B or b1_cell_info_L≟D or b1_cell_info_L≟d or A_Prepos_l[A_VL1]≟p[0,0,0,0,0,0]"
                      if (b1_cell_info_L == B  or  b1_cell_info_L == D  or  b1_cell_info_L == d  or  A_Prepos_l[A_VL1] == p[0,0,0,0,0,0]):
                        $ 408 "write_port_register(touch_cell_155,5)"
                        write_port_register(touch_cell_155,5)
                        $ 409 "write_port_register(touch_num_156,2)"
                        write_port_register(touch_num_156,2)
                        $ 410 "Call touch_sub"
                        touch_sub()
                        $ 411 "g_cp≔get_actual_tcp_pose()"
                        global g_cp= get_actual_tcp_pose ()
                        $ 412 "If g_cp[2]<(get_margin_z+a7_cell_bottom)/1000"
                        if (g_cp[2]<(get_margin_z+a7_cell_bottom)/1000):
                          $ 413 "g_cp[2]=(get_margin_z+a7_cell_bottom)/1000"
                          g_cp[2]=(get_margin_z+a7_cell_bottom)/1000
                        end
                        $ 414 "A_Prepos_l[move_i]=g_cp"
                        A_Prepos_l[move_i]=g_cp
                      end
                    else:
                      $ 415 "ElseIf move_i≟A_HOR_MR"
                      if (move_i == A_HOR_MR):
                        $ 416 "If b1_cell_info_L≟B or b1_cell_info_L≟D or b1_cell_info_L≟d or A_Prepos_l[A_VL1]≟p[0,0,0,0,0,0]"
                        if (b1_cell_info_L == B  or  b1_cell_info_L == D  or  b1_cell_info_L == d  or  A_Prepos_l[A_VL1] == p[0,0,0,0,0,0]):
                          $ 417 "write_port_register(touch_cell_155,5)"
                          write_port_register(touch_cell_155,5)
                          $ 418 "write_port_register(touch_num_156,4)"
                          write_port_register(touch_num_156,4)
                          $ 419 "Call touch_sub"
                          touch_sub()
                          $ 420 "g_cp≔get_actual_tcp_pose()"
                          global g_cp= get_actual_tcp_pose ()
                          $ 421 "If g_cp[2]<(get_margin_z+a7_cell_bottom)/1000"
                          if (g_cp[2]<(get_margin_z+a7_cell_bottom)/1000):
                            $ 422 "g_cp[2]=(get_margin_z+a7_cell_bottom)/1000"
                            g_cp[2]=(get_margin_z+a7_cell_bottom)/1000
                          end
                          $ 423 "A_Prepos_l[move_i]=g_cp"
                          A_Prepos_l[move_i]=g_cp
                        end
                      else:
                        $ 424 "Else" "noBreak"
                        $ 425 "write_port_register(touch_cell_155,move_i)"
                        write_port_register(touch_cell_155,move_i)
                        $ 426 "write_port_register(touch_num_156,1)"
                        write_port_register(touch_num_156,1)
                        $ 427 "Call touch_sub"
                        touch_sub()
                        $ 428 "A_Prepos_l[move_i]=get_actual_tcp_pose()"
                        A_Prepos_l[move_i]= get_actual_tcp_pose ()
                        $ 429 "If move_i≤4"
                        if (move_i <= 4):
                          $ 430 "write_port_register(touch_cell_155,move_i)"
                          write_port_register(touch_cell_155,move_i)
                          $ 431 "write_port_register(touch_num_156,2)"
                          write_port_register(touch_num_156,2)
                          $ 432 "Wait: 0.1"
                          sleep(0.1)
                          $ 433 "Call touch_sub"
                          touch_sub()
                          $ 434 "A_Prepos_l[move_i+9]=get_actual_tcp_pose()"
                          A_Prepos_l[move_i+9]= get_actual_tcp_pose ()
                        end
                      end
                    end
                  end
                end
              else:
                $ 435 "Else" "noBreak"
                $ 436 "A_Prepos_l[move_i]=p[0,0,0,0,0,0]"
                A_Prepos_l[move_i]=p[0,0,0,0,0,0]
                $ 437 "If move_i≤4"
                if (move_i <= 4):
                  $ 438 "A_Prepos_l[move_i+7]=p[0,0,0,0,0,0]"
                  A_Prepos_l[move_i+7]=p[0,0,0,0,0,0]
                else:
                  $ 439 "ElseIf move_i≟A_HOR"
                  if (move_i == A_HOR):
                    $ 440 "A_Prepos_l[A_HOR_ML]=p[0,0,0,0,0,0]"
                    A_Prepos_l[A_HOR_ML]=p[0,0,0,0,0,0]
                    $ 441 "A_Prepos_l[A_HOR_MR]=p[0,0,0,0,0,0]"
                    A_Prepos_l[A_HOR_MR]=p[0,0,0,0,0,0]
                    $ 442 "A_Prepos_l[A_HOR_M]=p[0,0,0,0,0,0]"
                    A_Prepos_l[A_HOR_M]=p[0,0,0,0,0,0]
                    $ 443 "A_Prepos_l[A_HOR_R]=p[0,0,0,0,0,0]"
                    A_Prepos_l[A_HOR_R]=p[0,0,0,0,0,0]
                  end
                end
              end
              $ 444 "move_i≔move_i+1"
              global move_i=move_i+1
            end
            $ 445 "change deg"
            $ 446 "move_i≔1"
            global move_i=1
            $ 447 "Loop move_i<14"
            while (move_i<14):
              $ 448 "If A_Prepos_l[move_i]≠p[0,0,0,0,0,0]"
              if (A_Prepos_l[move_i] != p[0,0,0,0,0,0]):
                $ 449 "If move_i≟A_VL1 or move_i≟A_VL2 or move_i≟A_VL1_END or move_i≟A_VL2_END"
                if (move_i == A_VL1  or  move_i == A_VL2  or  move_i == A_VL1_END  or  move_i == A_VL2_END):
                  $ 450 "b2_left_par≔ True "
                  global b2_left_par=  True
                  $ 451 "b8_wv_2f≔ False "
                  global b8_wv_2f=  False
                  $ 452 "get_pos≔A_Prepos_l[move_i]"
                  global get_pos=A_Prepos_l[move_i]
                  $ 453 "get_org≔left"
                  global get_org=p[.480496318984, .411279115151, .006998291210, -2.211681476386, -.899147924387, -1.383032568605]
                  $ 454 "get_pos≔p[get_pos[0],get_pos[1],get_pos[2],get_org[3],get_org[4],get_org[5]]"
                  global get_pos=p[get_pos[0],get_pos[1],get_pos[2],get_org[3],get_org[4],get_org[5]]
                  $ 455 "pre_tp≔tilt_3f_fun(get_pos,[0,0],a5_f_hole[1])"
                  global pre_tp=tilt_3f_fun(get_pos,[0,0],a5_f_hole[1])
                else:
                  $ 456 "ElseIf move_i≟A_VR1 or move_i≟A_VR2 or move_i≟A_VR1_END or move_i≟A_VR2_END"
                  if (move_i == A_VR1  or  move_i == A_VR2  or  move_i == A_VR1_END  or  move_i == A_VR2_END):
                    $ 457 "b2_left_par≔ False "
                    global b2_left_par=  False
                    $ 458 "b8_wv_2f≔ False "
                    global b8_wv_2f=  False
                    $ 459 "get_pos≔A_Prepos_l[move_i]"
                    global get_pos=A_Prepos_l[move_i]
                    $ 460 "get_org≔right"
                    global get_org=p[.475000000000, -.421403215678, .026417194146, 1.917761036827, -1.141682393512, 1.523356199292]
                    $ 461 "get_pos≔p[get_pos[0],get_pos[1],get_pos[2],get_org[3],get_org[4],get_org[5]]"
                    global get_pos=p[get_pos[0],get_pos[1],get_pos[2],get_org[3],get_org[4],get_org[5]]
                    $ 462 "pre_tp≔tilt_3f_fun(get_pos,[0,0],a5_f_hole[1])"
                    global pre_tp=tilt_3f_fun(get_pos,[0,0],a5_f_hole[1])
                  else:
                    $ 463 "ElseIf move_i≟A_HOR or move_i≟A_HOR_ML"
                    if (move_i == A_HOR  or  move_i == A_HOR_ML):
                      $ 464 "b8_wv_2f≔ True "
                      global b8_wv_2f=  True
                      $ 465 "b2_left_par≔ True "
                      global b2_left_par=  True
                      $ 466 "get_pos≔A_Prepos_l[move_i]"
                      global get_pos=A_Prepos_l[move_i]
                      $ 467 "get_org≔up_left"
                      global get_org=p[.492775857339, .409517380626, -.029063830209, -2.419264859926, -.998084331190, -1.368689080860]
                      $ 468 "get_pos≔p[get_pos[0],get_pos[1],get_pos[2],get_org[3],get_org[4],get_org[5]]"
                      global get_pos=p[get_pos[0],get_pos[1],get_pos[2],get_org[3],get_org[4],get_org[5]]
                      $ 469 "pre_tp≔tilt_2f_fun(get_pos,[0,0], True , True )"
                      global pre_tp=tilt_2f_fun(get_pos,[0,0],  True  ,  True  )
                    else:
                      $ 470 "ElseIf move_i≟A_HOR_R or move_i≟A_HOR_MR"
                      if (move_i == A_HOR_R  or  move_i == A_HOR_MR):
                        $ 471 "b8_wv_2f≔ True "
                        global b8_wv_2f=  True
                        $ 472 "b2_left_par≔ False "
                        global b2_left_par=  False
                        $ 473 "get_pos≔A_Prepos_l[move_i]"
                        global get_pos=A_Prepos_l[move_i]
                        $ 474 "get_org≔up_right"
                        global get_org=p[.445203173045, -.406687378356, -.031125942276, 2.308490741423, -1.066468937023, 1.322151316133]
                        $ 475 "get_pos≔p[get_pos[0],get_pos[1],get_pos[2],get_org[3],get_org[4],get_org[5]]"
                        global get_pos=p[get_pos[0],get_pos[1],get_pos[2],get_org[3],get_org[4],get_org[5]]
                        $ 476 "pre_tp≔tilt_2f_fun(get_pos,[0,0], False , True )"
                        global pre_tp=tilt_2f_fun(get_pos,[0,0],  False  ,  True  )
                      end
                    end
                  end
                end
                $ 477 "A_Prepos_l[move_i]=pre_tp"
                A_Prepos_l[move_i]=pre_tp
              end
              $ 478 "move_i≔move_i+1"
              global move_i=move_i+1
            end
            $ 479 "homeing()"
            homeing()
            $ 480 "Wait read_port_register(170)≟1"
            while (not( read_port_register (170) == 1)):
              sync()
            end
            $ 481 "write_port_register(170,0)"
            write_port_register(170,0)
          else:
            $ 482 "Else" "noBreak"
            $ 483 "value from pendant"
            $ 484 "move_i≔1"
            global move_i=1
            $ 486 "Touch_FrontandSide"
            $ 487 "If EXT_flag1[11]≟ True "
            if (EXT_flag1[11] ==   True  ):
              $ 488 "Touch front and side_Right"
              $ 489 "move_center≔pose_add(first_p_wp, p[-first_p_wp[0]+(get_center-work_touch_dis)/1000,0,0,0,0,0])"
              global move_center= pose_add (first_p_wp, p[-first_p_wp[0]+(get_center-work_touch_dis)/1000,0,0,0,0,0])
              $ 490 "get_pose_side_t≔0"
              global get_pose_side_t=0
              $ 492 "move_center[2]=(center_height+a7_cell_bottom)/1000"
              move_center[2]=(center_height+a7_cell_bottom)/1000
              $ 494 "MoveL"
              $ 495 "move_center" "breakAfter"
              movel(pose_trans(Base, move_center), a=0.5, v=0.15)
              $ 496 "touch_center≔contact_fun(p[0,0,0,0,0,0],[1,0,0],20000,20,20)"
              global touch_center=contact_fun(p[0,0,0,0,0,0],[1,0,0],20000,20,20)
              $ 497 "direction(p[0,0,0,0,0,0],[-1,0,0],10,180,200)"
              direction(p[0,0,0,0,0,0],[-1,0,0],10,180,200)
              $ 498 "get_center≔touch_center[0]*1000"
              global get_center=touch_center[0]*1000
              $ 499 "a7_f_distance≔get_center"
              global a7_f_distance=get_center
              $ 500 "move_center≔pose_add(move_center,p[0,sec_touch_dis/1000,0,0,0,0])"
              global move_center= pose_add (move_center,p[0,sec_touch_dis/1000,0,0,0,0])
              $ 501 "move_center[0]=touch_center[0]-20/1000"
              move_center[0]=touch_center[0]-20/1000
              $ 502 "MoveL"
              $ 503 "move_center" "breakAfter"
              movel(pose_trans(Base, move_center), a=0.5, v=0.15)
              $ 504 "touch_center2≔contact_fun(p[0,0,0,0,0,0],[1,0,0],20000,20,20)"
              global touch_center2=contact_fun(p[0,0,0,0,0,0],[1,0,0],20000,20,20)
              $ 505 "center_line≔get_feature_Line(touch_center,touch_center2)"
              global center_line=get_feature_Line(touch_center,touch_center2)
              $ 506 "event_cal_on≔ True "
              global event_cal_on=  True
              $ 507 "direction(p[0,0,0,0,0,0],[-1,0,0],10,180,200)"
              direction(p[0,0,0,0,0,0],[-1,0,0],10,180,200)
              $ 509 "homeing()"
              homeing()
              $ 510 "b2_left_par≔ False "
              global b2_left_par=  False
              $ 511 "b8_wv_2f≔ False "
              global b8_wv_2f=  False
              $ 512 "b2_cell≔b1_cell_info_R"
              global b2_cell=b1_cell_info_R
              $ 513 "get_pos≔get_lr(side_p_R,a6_f_width,[35,0,0,0,0],a7_f_distance,b2_left_par,b8_wv_2f,Touch_dis,get_margin_z,get_pose_side_t,30,0,center_line, True )"
              global get_pos=get_lr(p[.471584857321, -.427242166643, .026448165242, 1.806736638758, -1.227818761912, 1.383474453522],a6_f_width,[35,0,0,0,0],a7_f_distance,b2_left_par,b8_wv_2f,Touch_dis,get_margin_z,get_pose_side_t,30,0,center_line,  True  )
              $ 515 "pre_tp≔get_pos"
              global pre_tp=get_pos
              $ 516 "pre_tp≔pose_add(pre_tp, p[side_pos_x/1000,0,0,0,0,0])"
              global pre_tp= pose_add (pre_tp, p[side_pos_x/1000,0,0,0,0,0])
              $ 517 "pre_tp[2]=(center_height+a7_cell_bottom)/1000"
              pre_tp[2]=(center_height+a7_cell_bottom)/1000
              $ 518 "MoveL"
              $ 519 "pre_tp" "breakAfter"
              movel(pose_trans(Base, pre_tp), a=0.8, v=0.4)
              $ 520 "touch_side≔contact_fun(p[0,0,0,0,0,0],[0,-1,0],20000,13,13)"
              global touch_side=contact_fun(p[0,0,0,0,0,0],[0,-1,0],20000,13,13)
              $ 521 "touch_side≔get_feature_pose(touch_side,center_line)"
              global touch_side=get_feature_pose(touch_side,center_line)
              $ 522 "direction(p[0,0,0,0,0,0],[0,1,0],10,180,200)"
              direction(p[0,0,0,0,0,0],[0,1,0],10,180,200)
              $ 523 "write_welder(4, False )"
              write_welder(4,  False  )
              $ 524 "get_pose_side_t≔touch_side[1]*1000"
              global get_pose_side_t=touch_side[1]*1000
              $ 525 "get_pose_side_t≔get_pose_side_t+(a6_f_width/2)"
              global get_pose_side_t=get_pose_side_t+(a6_f_width/2)
              $ 526 "event_side_on≔ True "
              global event_side_on=  True
              $ 527 "MoveL"
              $ 528 "Direction: Base"
              global move_thread_flag_528=0
              thread move_thread_528():
                enter_critical
                move_thread_flag_528 = 1
                local towardsPos=calculate_point_to_move_towards(p[0.0,0.0,0.0,0.0,0.0,0.0], [-1,1,0], 0.03)
                movel(towardsPos, a=0.3, v=0.15)
                move_thread_flag_528 = 2
                exit_critical
              end
              move_thread_flag_528 = 0
              move_thread_han_528 = run move_thread_528()
              while (True):
                sleep(1.0E-10)
                if (move_thread_flag_528 > 1):
                  join move_thread_han_528
                  $ 529 "Until (distance)"
                  break
                end
                sync()
              end
              $ 530 "homeing()"
              homeing()
            else:
              $ 531 "Else" "noBreak"
              $ 532 "Touch front and side_Left"
              $ 533 "move_center≔pose_add(first_p_wp, p[-first_p_wp[0]+(get_center-work_touch_dis)/1000,0,0,0,0,0])"
              global move_center= pose_add (first_p_wp, p[-first_p_wp[0]+(get_center-work_touch_dis)/1000,0,0,0,0,0])
              $ 534 "get_pose_side_t≔0"
              global get_pose_side_t=0
              $ 536 "move_center[2]=(center_height+a7_cell_bottom)/1000"
              move_center[2]=(center_height+a7_cell_bottom)/1000
              $ 538 "MoveL"
              $ 539 "move_center" "breakAfter"
              movel(pose_trans(Base, move_center), a=0.5, v=0.15)
              $ 540 "touch_center≔contact_fun(p[0,0,0,0,0,0],[1,0,0],20000,20,20)"
              global touch_center=contact_fun(p[0,0,0,0,0,0],[1,0,0],20000,20,20)
              $ 541 "direction(p[0,0,0,0,0,0],[-1,0,0],10,180,200)"
              direction(p[0,0,0,0,0,0],[-1,0,0],10,180,200)
              $ 542 "get_center≔touch_center[0]*1000"
              global get_center=touch_center[0]*1000
              $ 543 "a7_f_distance≔get_center"
              global a7_f_distance=get_center
              $ 544 "move_center≔pose_add(move_center,p[0,sec_touch_dis/1000,0,0,0,0])"
              global move_center= pose_add (move_center,p[0,sec_touch_dis/1000,0,0,0,0])
              $ 545 "move_center[0]=touch_center[0]-20/1000"
              move_center[0]=touch_center[0]-20/1000
              $ 546 "MoveL"
              $ 547 "move_center" "breakAfter"
              movel(pose_trans(Base, move_center), a=0.5, v=0.15)
              $ 548 "touch_center2≔contact_fun(p[0,0,0,0,0,0],[1,0,0],20000,20,20)"
              global touch_center2=contact_fun(p[0,0,0,0,0,0],[1,0,0],20000,20,20)
              $ 549 "center_line≔get_feature_Line(touch_center,touch_center2)"
              global center_line=get_feature_Line(touch_center,touch_center2)
              $ 550 "event_cal_on≔ True "
              global event_cal_on=  True
              $ 551 "direction(p[0,0,0,0,0,0],[-1,0,0],10,180,200)"
              direction(p[0,0,0,0,0,0],[-1,0,0],10,180,200)
              $ 553 "homeing()"
              homeing()
              $ 554 "b2_left_par≔ True "
              global b2_left_par=  True
              $ 555 "b8_wv_2f≔ False "
              global b8_wv_2f=  False
              $ 556 "b2_cell≔b1_cell_info_L"
              global b2_cell=b1_cell_info_L
              $ 557 "get_pos≔get_lr(side_p_L,a6_f_width,[35,0,0,0,0],a7_f_distance,b2_left_par,b8_wv_2f,Touch_dis,get_margin_z,get_pose_side_t,30,0,center_line, True )"
              global get_pos=get_lr(p[.411215372122, .375785944375, -.010176539343, -1.953488355698, -1.125710367676, -1.228829273458],a6_f_width,[35,0,0,0,0],a7_f_distance,b2_left_par,b8_wv_2f,Touch_dis,get_margin_z,get_pose_side_t,30,0,center_line,  True  )
              $ 559 "pre_tp≔get_pos"
              global pre_tp=get_pos
              $ 560 "pre_tp≔pose_add(pre_tp, p[side_pos_x/1000,0,0,0,0,0])"
              global pre_tp= pose_add (pre_tp, p[side_pos_x/1000,0,0,0,0,0])
              $ 561 "pre_tp[2]=(center_height+a7_cell_bottom)/1000"
              pre_tp[2]=(center_height+a7_cell_bottom)/1000
              $ 562 "MoveL"
              $ 563 "pre_tp" "breakAfter"
              movel(pose_trans(Base, pre_tp), a=0.8, v=0.4)
              $ 564 "touch_side≔contact_fun(p[0,0,0,0,0,0],[0,1,0],20000,13,13)"
              global touch_side=contact_fun(p[0,0,0,0,0,0],[0,1,0],20000,13,13)
              $ 565 "touch_side≔get_feature_pose(touch_side,center_line)"
              global touch_side=get_feature_pose(touch_side,center_line)
              $ 566 "direction(p[0,0,0,0,0,0],[0,-1,0],10,180,200)"
              direction(p[0,0,0,0,0,0],[0,-1,0],10,180,200)
              $ 567 "write_welder(4, False )"
              write_welder(4,  False  )
              $ 568 "get_pose_side_t≔touch_side[1]*1000"
              global get_pose_side_t=touch_side[1]*1000
              $ 569 "get_pose_side_t≔get_pose_side_t-(a6_f_width/2)"
              global get_pose_side_t=get_pose_side_t-(a6_f_width/2)
              $ 570 "event_side_on≔ True "
              global event_side_on=  True
              $ 571 "MoveL"
              $ 572 "Direction: Base"
              global move_thread_flag_572=0
              thread move_thread_572():
                enter_critical
                move_thread_flag_572 = 1
                local towardsPos=calculate_point_to_move_towards(p[0.0,0.0,0.0,0.0,0.0,0.0], [-1,-1,0], 0.03)
                movel(towardsPos, a=0.3, v=0.15)
                move_thread_flag_572 = 2
                exit_critical
              end
              move_thread_flag_572 = 0
              move_thread_han_572 = run move_thread_572()
              while (True):
                sleep(1.0E-10)
                if (move_thread_flag_572 > 1):
                  join move_thread_han_572
                  $ 573 "Until (distance)"
                  break
                end
                sync()
              end
              $ 574 "homeing()"
              homeing()
            end
            $ 576 "Wait event_side_on≟ False "
            while (not(event_side_on ==   False  )):
              sync()
            end
          end
          $ 577 "move and touch"
          $ 578 "Touch Move"
          $ 579 "HOR_L"
          $ 580 "If A_Prepos_l[A_HOR]≠p[0,0,0,0,0,0]"
          if (A_Prepos_l[A_HOR] != p[0,0,0,0,0,0]):
            $ 581 "b2_left_par≔ True "
            global b2_left_par=  True
            $ 582 "b8_wv_2f≔ True "
            global b8_wv_2f=  True
            $ 583 "b7_tilt_degree≔[0,0,0]"
            global b7_tilt_degree=[0,0,0]
            $ 584 "A_sel_v≔A_HOR"
            global A_sel_v=A_HOR
            $ 585 "wv_direction≔1"
            global wv_direction=1
            $ 586 "Call MoveandTouchFun_2f"
            MoveandTouchFun_2f()
            $ 588 "If b1_cell_info_L≟A or b1_cell_info_L≟C or b1_cell_info_L≟c"
            if (b1_cell_info_L == A  or  b1_cell_info_L == C  or  b1_cell_info_L == c):
              $ 589 "If A_Prepos_l[A_VL1]≟p[0,0,0,0,0,0]"
              if (A_Prepos_l[A_VL1] == p[0,0,0,0,0,0]):
                $ 591 "g_tp≔A_Prepos_l[A_HOR]"
                global g_tp=A_Prepos_l[A_HOR]
                $ 594 "Folder"
                $ 595 "g_cp≔get_actual_tcp_pose()"
                global g_cp= get_actual_tcp_pose ()
                $ 596 "g_cp≔pose_trans(g_cp, p[0,0,0,d2r(12),d2r(5),0])"
                global g_cp= pose_trans (g_cp, p[0,0,0,d2r(12),d2r(5),0])
                $ 597 "MoveL"
                $ 598 "g_cp" "breakAfter"
                movel(pose_trans(Base, g_cp), a=0.08, v=0.08)
                $ 599 "for_x_HOR≔contact_fun(A_Touch_p[A_sel_v],[-1*wv_direction,0,0],10000,15,15,  False)"
                global for_x_HOR=contact_fun(A_Touch_p[A_sel_v],[-1*wv_direction,0,0],10000,15,15,  False)
                $ 600 "direction(p[0,0,0,0,0,0],[0,-1,0],20,120,160)"
                direction(p[0,0,0,0,0,0],[0,-1,0],20,120,160)
                $ 601 "write_welder(4, False )"
                write_welder(4,  False  )
              else:
                $ 602 "Else" "noBreak"
                $ 603 "for_x_HOR≔p[0,0,0,0,0,0]"
                global for_x_HOR=p[0,0,0,0,0,0]
              end
            else:
              $ 604 "ElseIf b1_cell_info_L≟E"
              if (b1_cell_info_L == E):
                $ 605 "direction(p[0,0,0,0,0,0],[0,1,0],40,120,160)"
                direction(p[0,0,0,0,0,0],[0,1,0],40,120,160)
                $ 606 "direction(p[0,0,0,0,0,0],[1,0,0],20,120,160)"
                direction(p[0,0,0,0,0,0],[1,0,0],20,120,160)
                $ 607 "for_x_HOR≔contact_fun(A_Touch_p[A_sel_v],[0,-1,0],10000,15,15,  False)"
                global for_x_HOR=contact_fun(A_Touch_p[A_sel_v],[0,-1,0],10000,15,15,  False)
                $ 608 "write_welder(4, False )"
                write_welder(4,  False  )
                $ 609 "direction(p[0,0,0,0,0,0],[0,1,0],20,120,160)"
                direction(p[0,0,0,0,0,0],[0,1,0],20,120,160)
                $ 610 "direction(p[0,0,0,0,0,0],[-1,0,0],40,120,160)"
                direction(p[0,0,0,0,0,0],[-1,0,0],40,120,160)
              end
            end
            $ 611 "If point_dist(A_Prepos_l[A_HOR], A_Prepos_l[A_VL1])>0.032"
            if (point_dist(A_Prepos_l[A_HOR], A_Prepos_l[A_VL1])>0.032):
              $ 612 "homeing()"
              homeing()
            end
          end
          $ 613 "VL1"
          $ 614 "If A_Prepos_l[A_VL1]≠p[0,0,0,0,0,0]"
          if (A_Prepos_l[A_VL1] != p[0,0,0,0,0,0]):
            $ 615 "b2_left_par≔ True "
            global b2_left_par=  True
            $ 616 "b8_wv_2f≔ False "
            global b8_wv_2f=  False
            $ 617 "b7_tilt_degree≔[0,0,0]"
            global b7_tilt_degree=[0,0,0]
            $ 618 "A_sel_v≔A_VL1"
            global A_sel_v=A_VL1
            $ 619 "A_sel_v_end≔A_VL1_END"
            global A_sel_v_end=A_VL1_END
            $ 620 "b2_par_cd≔0"
            global b2_par_cd=0
            $ 621 "If b1_cell_info_L≟A or b1_cell_info_L≟C or b1_cell_info_L≟c"
            if (b1_cell_info_L == A  or  b1_cell_info_L == C  or  b1_cell_info_L == c):
              $ 622 "Scallup_check≔ True "
              global Scallup_check=  True
            else:
              $ 623 "Else" "noBreak"
              $ 624 "Scallup_check≔ False "
              global Scallup_check=  False
            end
            $ 625 "Call MoveandTouchFun_3f"
            MoveandTouchFun_3f()
            $ 626 "If b1_cell_info_L≟A or b1_cell_info_L≟C or b1_cell_info_L≟c"
            if (b1_cell_info_L == A  or  b1_cell_info_L == C  or  b1_cell_info_L == c):
              $ 627 "If A_Prepos_l[A_HOR]≟p[0,0,0,0,0,0]"
              if (A_Prepos_l[A_HOR] == p[0,0,0,0,0,0]):
                $ 628 "direction(p[0,0,0,0,0,0],[0,-1,0],8,120,160)"
                direction(p[0,0,0,0,0,0],[0,-1,0],8,120,160)
                $ 630 "AAgcp≔get_actual_tcp_pose()"
                global AAgcp= get_actual_tcp_pose ()
                $ 631 "AAgangle≔up_left"
                global AAgangle=p[.492775857339, .409517380626, -.029063830209, -2.419264859926, -.998084331190, -1.368689080860]
                $ 632 "AAgtp≔p[AAgcp[0],AAgcp[1],AAgcp[2],AAgangle[3],AAgangle[4],AAgangle[5]]"
                global AAgtp=p[AAgcp[0],AAgcp[1],AAgcp[2],AAgangle[3],AAgangle[4],AAgangle[5]]
                $ 633 "MoveL"
                $ 634 "AAgtp" "breakAfter"
                movel(pose_trans(Base, AAgtp), a=0.08, v=0.08)
                $ 636 "for_z_VL1≔contact_fun(p[0,0,0,0,0,0],[0,0,-1],10000,15,15,  False)"
                global for_z_VL1=contact_fun(p[0,0,0,0,0,0],[0,0,-1],10000,15,15,  False)
                $ 637 "direction(p[0,0,0,0,0,0],[0,0,1],20,120,160)"
                direction(p[0,0,0,0,0,0],[0,0,1],20,120,160)
                $ 638 "write_welder(4, False )"
                write_welder(4,  False  )
              else:
                $ 639 "Else" "noBreak"
                $ 640 "for_z_VL1≔p[0,0,0,0,0,0]"
                global for_z_VL1=p[0,0,0,0,0,0]
              end
            end
          end
          $ 641 "HOR_ML"
          $ 642 "If A_Prepos_l[A_HOR_ML]≠p[0,0,0,0,0,0]"
          if (A_Prepos_l[A_HOR_ML] != p[0,0,0,0,0,0]):
            $ 643 "b2_left_par≔ True "
            global b2_left_par=  True
            $ 644 "b8_wv_2f≔ True "
            global b8_wv_2f=  True
            $ 645 "b7_tilt_degree≔[0,0,0]"
            global b7_tilt_degree=[0,0,0]
            $ 646 "A_sel_v≔A_HOR_ML"
            global A_sel_v=A_HOR_ML
            $ 647 "If b1_cell_info_L≟C or b1_cell_info_L≟D"
            if (b1_cell_info_L == C  or  b1_cell_info_L == D):
              $ 648 "wv_direction≔1"
              global wv_direction=1
              $ 649 "Call MoveFun"
              MoveFun()
              $ 650 "for_cal_xy≔contact_fun(p[0,0,0,0,0,0],[1,0,0],20000,20,20)"
              global for_cal_xy=contact_fun(p[0,0,0,0,0,0],[1,0,0],20000,20,20)
              $ 651 "direction(p[0,0,0,0,0,0],[-1,0,0],15,120,160)"
              direction(p[0,0,0,0,0,0],[-1,0,0],15,120,160)
              $ 652 "direction(p[0,0,0,0,0,0],[0,-1,0],60,120,160)"
              direction(p[0,0,0,0,0,0],[0,-1,0],60,120,160)
              $ 653 "direction(p[0,0,0,0,0,0],[1,0,0],20,120,160)"
              direction(p[0,0,0,0,0,0],[1,0,0],20,120,160)
              $ 654 "for_cal_x_wel≔contact_fun(p[0,0,0,0,0,0],[0,1,0],20000,20,20)"
              global for_cal_x_wel=contact_fun(p[0,0,0,0,0,0],[0,1,0],20000,20,20)
              $ 655 "direction(p[0,0,0,0,0,0],[0,-1,0],20,120,160)"
              direction(p[0,0,0,0,0,0],[0,-1,0],20,120,160)
              $ 656 "for_cal_zl≔contact_fun(p[0,0,0,0,0,0],[0,0,-1],20000,20,20)"
              global for_cal_zl=contact_fun(p[0,0,0,0,0,0],[0,0,-1],20000,20,20)
              $ 657 "direction(p[0,0,0,0,0,0],[0,0,1],20,120,160)"
              direction(p[0,0,0,0,0,0],[0,0,1],20,120,160)
              $ 658 "If A_Prepos_l[A_VL2]≟p[0,0,0,0,0,0]"
              if (A_Prepos_l[A_VL2] == p[0,0,0,0,0,0]):
                $ 659 "for_cal_y_wel≔contact_fun(p[0,0,0,0,0,0],[1,0,0],20000,20,20)"
                global for_cal_y_wel=contact_fun(p[0,0,0,0,0,0],[1,0,0],20000,20,20)
                $ 660 "direction(p[0,0,0,0,0,0],[-1,0,0],30,120,160)"
                direction(p[0,0,0,0,0,0],[-1,0,0],30,120,160)
              end
              $ 661 "for_cal_rot≔A_Touch_p[A_HOR]"
              global for_cal_rot=A_Touch_p[A_HOR]
              $ 662 "A_Touch_p[A_sel_v]=p[for_cal_xy[0],for_cal_xy[1],for_cal_zl[2],for_cal_rot[3],for_cal_rot[4],for_cal_rot[5]]"
              A_Touch_p[A_sel_v]=p[for_cal_xy[0],for_cal_xy[1],for_cal_zl[2],for_cal_rot[3],for_cal_rot[4],for_cal_rot[5]]
              $ 663 "A_Touch_p[A_sel_v]=pose_trans(A_Touch_p[A_sel_v], p[Touch_dis/1000,0,0,0,0,0])"
              A_Touch_p[A_sel_v]= pose_trans (A_Touch_p[A_sel_v], p[Touch_dis/1000,0,0,0,0,0])
              $ 664 "write_welder(4, False )"
              write_welder(4,  False  )
            else:
              $ 665 "Else" "noBreak"
              $ 666 "wv_direction≔1"
              global wv_direction=1
              $ 667 "for_cal_rot≔A_Touch_p[A_HOR]"
              global for_cal_rot=A_Touch_p[A_HOR]
              $ 668 "Call MoveFun_cd"
              MoveFun_cd()
              $ 669 "for_cal_y_wel≔contact_fun(p[0,0,0,0,0,0],[1,0,0],20000,20,20)"
              global for_cal_y_wel=contact_fun(p[0,0,0,0,0,0],[1,0,0],20000,20,20)
              $ 670 "for_cal_y_wel[2]=for_cal_rot[2]"
              for_cal_y_wel[2]=for_cal_rot[2]
              $ 671 "dir_x_cal≔get_feature_Line(for_cal_rot,for_cal_y_wel)"
              global dir_x_cal=get_feature_Line(for_cal_rot,for_cal_y_wel)
              $ 672 "direction(p[0,0,0,0,0,0],[-1,0,0],40,120,160)"
              direction(p[0,0,0,0,0,0],[-1,0,0],40,120,160)
              $ 673 "direction(p[0,0,0,0,0,0],[0,-1,0],80,120,160)"
              direction(p[0,0,0,0,0,0],[0,-1,0],80,120,160)
              $ 674 "for_cal_y_wel≔contact_fun(p[0,0,0,0,0,0],[1,0,0],20000,20,20)"
              global for_cal_y_wel=contact_fun(p[0,0,0,0,0,0],[1,0,0],20000,20,20)
              $ 675 "direction(p[0,0,0,0,0,0],[-1,0,0],5,120,160)"
              direction(p[0,0,0,0,0,0],[-1,0,0],5,120,160)
              $ 676 "direction(p[0,0,0,0,0,0],[0,1,0],50,120,160)"
              direction(p[0,0,0,0,0,0],[0,1,0],50,120,160)
              $ 677 "direction(p[0,0,0,0,0,0],[1,0,0],7,120,160)"
              direction(p[0,0,0,0,0,0],[1,0,0],7,120,160)
              $ 678 "for_cal_x_wel≔contact_fun(p[0,0,0,0,0,0],[0,-1,0],20000,20,20)"
              global for_cal_x_wel=contact_fun(p[0,0,0,0,0,0],[0,-1,0],20000,20,20)
              $ 679 "get_ml≔get_feature_pose(for_cal_x_wel,for_cal_rot)"
              global get_ml=get_feature_pose(for_cal_x_wel,for_cal_rot)
              $ 681 "A_Touch_p[A_sel_v]=feature_offset(for_cal_rot,p[0,get_ml[0]+(-cd_offset+cd_extra_dis)/1000,0,0,0,0],dir_x_cal)"
              A_Touch_p[A_sel_v]=feature_offset(for_cal_rot,p[0,get_ml[0]+(-cd_offset+cd_extra_dis)/1000,0,0,0,0],dir_x_cal)
              $ 682 "direction(p[0,0,0,0,0,0],[0,1,0],5,120,160)"
              direction(p[0,0,0,0,0,0],[0,1,0],5,120,160)
              $ 683 "direction(p[0,0,0,0,0,0],[-1,0,0],20,120,160)"
              direction(p[0,0,0,0,0,0],[-1,0,0],20,120,160)
              $ 684 "write_welder(4, False )"
              write_welder(4,  False  )
            end
          else:
            $ 685 "Else" "noBreak"
            $ 686 "homeing()"
            homeing()
          end
          $ 687 "VL2"
          $ 688 "If A_Prepos_l[A_VL2]≠p[0,0,0,0,0,0]"
          if (A_Prepos_l[A_VL2] != p[0,0,0,0,0,0]):
            $ 689 "b2_left_par≔ True "
            global b2_left_par=  True
            $ 690 "b8_wv_2f≔ False "
            global b8_wv_2f=  False
            $ 691 "b7_tilt_degree≔basic_tilt_3f"
            global b7_tilt_degree=basic_tilt_3f
            $ 692 "A_sel_v≔A_VL2"
            global A_sel_v=A_VL2
            $ 693 "A_sel_v_end≔A_VL2_END"
            global A_sel_v_end=A_VL2_END
            $ 694 "b2_par_cd≔1"
            global b2_par_cd=1
            $ 695 "If b1_cell_info_L≟A or b1_cell_info_L≟C or b1_cell_info_L≟c"
            if (b1_cell_info_L == A  or  b1_cell_info_L == C  or  b1_cell_info_L == c):
              $ 696 "Scallup_check≔ True "
              global Scallup_check=  True
            else:
              $ 697 "Else" "noBreak"
              $ 698 "Scallup_check≔ False "
              global Scallup_check=  False
            end
            $ 699 "If b1_cell_info_L≟d or b1_cell_info_L≟c"
            if (b1_cell_info_L == d  or  b1_cell_info_L == c):
              $ 700 "Halt"
              halt
            else:
              $ 701 "Else" "noBreak"
              $ 702 "If A_Touch_p[A_VL1]≟p[0,0,0,0,0,0]"
              if (A_Touch_p[A_VL1] == p[0,0,0,0,0,0]):
                $ 703 "Call MoveandTouchFun_3f"
                MoveandTouchFun_3f()
                $ 704 "If A_Prepos_l[A_HOR_ML]≟p[0,0,0,0,0,0]"
                if (A_Prepos_l[A_HOR_ML] == p[0,0,0,0,0,0]):
                  $ 705 "direction(p[0,0,0,0,0,0],[0,-1,0],8,120,160)"
                  direction(p[0,0,0,0,0,0],[0,-1,0],8,120,160)
                  $ 706 "AAgcp≔get_actual_tcp_pose()"
                  global AAgcp= get_actual_tcp_pose ()
                  $ 707 "AAgangle≔up_left"
                  global AAgangle=p[.492775857339, .409517380626, -.029063830209, -2.419264859926, -.998084331190, -1.368689080860]
                  $ 708 "AAgtp≔p[AAgcp[0],AAgcp[1],AAgcp[2],AAgangle[3],AAgangle[4],AAgangle[5]]"
                  global AAgtp=p[AAgcp[0],AAgcp[1],AAgcp[2],AAgangle[3],AAgangle[4],AAgangle[5]]
                  $ 709 "MoveL"
                  $ 710 "AAgtp" "breakAfter"
                  movel(pose_trans(Base, AAgtp), a=0.08, v=0.08)
                  $ 712 "for_cal_zl≔contact_fun(p[0,0,0,0,0,0],[0,0,-1],20000,20,20)"
                  global for_cal_zl=contact_fun(p[0,0,0,0,0,0],[0,0,-1],20000,20,20)
                end
                $ 713 "touch_tmp≔A_Touch_p[A_sel_v]"
                global touch_tmp=A_Touch_p[A_sel_v]
                $ 714 "touch_tmp[2]=for_cal_zl[2]"
                touch_tmp[2]=for_cal_zl[2]
                $ 715 "A_Touch_p[A_sel_v]=touch_tmp"
                A_Touch_p[A_sel_v]=touch_tmp
                $ 716 "for_cal_y_wel≔A_Touch_p[A_sel_v]"
                global for_cal_y_wel=A_Touch_p[A_sel_v]
                $ 717 "for_cal_x_wel≔A_Touch_p[A_sel_v]"
                global for_cal_x_wel=A_Touch_p[A_sel_v]
              else:
                $ 718 "Else" "noBreak"
                $ 719 "Call MoveFun"
                MoveFun()
                $ 720 "for_cal_y_wel≔contact_fun(p[0,0,0,0,0,0],[1,0,0],20000,20,20)"
                global for_cal_y_wel=contact_fun(p[0,0,0,0,0,0],[1,0,0],20000,20,20)
                $ 721 "direction(p[0,0,0,0,0,0],[-1,0,0],40,120,160)"
                direction(p[0,0,0,0,0,0],[-1,0,0],40,120,160)
                $ 722 "If A_Prepos_l[A_HOR_ML]≟p[0,0,0,0,0,0]"
                if (A_Prepos_l[A_HOR_ML] == p[0,0,0,0,0,0]):
                  $ 723 "direction(p[0,0,0,0,0,0],[0,1,0],60,120,160)"
                  direction(p[0,0,0,0,0,0],[0,1,0],60,120,160)
                  $ 724 "var_2≔contact_fun(p[0,0,0,0,0,0],[1,0,0],20000,20,20)"
                  global var_2=contact_fun(p[0,0,0,0,0,0],[1,0,0],20000,20,20)
                  $ 725 "direction(p[0,0,0,0,0,0],[-1,0,0],5,120,160)"
                  direction(p[0,0,0,0,0,0],[-1,0,0],5,120,160)
                  $ 726 "direction(p[0,0,0,0,0,0],[0,-1,0],60,120,160)"
                  direction(p[0,0,0,0,0,0],[0,-1,0],60,120,160)
                  $ 727 "direction(p[0,0,0,0,0,0],[1,0,0],10,120,160)"
                  direction(p[0,0,0,0,0,0],[1,0,0],10,120,160)
                  $ 728 "for_cal_x_wel≔contact_fun(p[0,0,0,0,0,0],[0,1,0],20000,20,20)"
                  global for_cal_x_wel=contact_fun(p[0,0,0,0,0,0],[0,1,0],20000,20,20)
                  $ 729 "direction(p[0,0,0,0,0,0],[0,-1,0],20,120,160)"
                  direction(p[0,0,0,0,0,0],[0,-1,0],20,120,160)
                  $ 730 "AAgcp≔get_actual_tcp_pose()"
                  global AAgcp= get_actual_tcp_pose ()
                  $ 731 "AAgangle≔up_left"
                  global AAgangle=p[.492775857339, .409517380626, -.029063830209, -2.419264859926, -.998084331190, -1.368689080860]
                  $ 732 "AAgtp≔p[AAgcp[0],AAgcp[1],AAgcp[2],AAgangle[3],AAgangle[4],AAgangle[5]]"
                  global AAgtp=p[AAgcp[0],AAgcp[1],AAgcp[2],AAgangle[3],AAgangle[4],AAgangle[5]]
                  $ 733 "MoveL"
                  $ 734 "AAgtp" "breakAfter"
                  movel(pose_trans(Base, AAgtp), a=0.08, v=0.08)
                  $ 736 "for_cal_zl≔contact_fun(p[0,0,0,0,0,0],[0,0,-1],20000,20,20)"
                  global for_cal_zl=contact_fun(p[0,0,0,0,0,0],[0,0,-1],20000,20,20)
                  $ 737 "direction(p[0,0,0,0,0,0],[0,0,1],10,120,160)"
                  direction(p[0,0,0,0,0,0],[0,0,1],10,120,160)
                  $ 738 "direction(p[0,0,0,0,0,0],[-1,0,0],20,120,160)"
                  direction(p[0,0,0,0,0,0],[-1,0,0],20,120,160)
                end
                $ 739 "for_cal_rot≔A_Touch_p[A_VL1]"
                global for_cal_rot=A_Touch_p[A_VL1]
                $ 740 "A_Touch_p[A_sel_v]=p[for_cal_y_wel[0],for_cal_x_wel[1],for_cal_zl[2],for_cal_rot[3],for_cal_rot[4],for_cal_rot[5]]"
                A_Touch_p[A_sel_v]=p[for_cal_y_wel[0],for_cal_x_wel[1],for_cal_zl[2],for_cal_rot[3],for_cal_rot[4],for_cal_rot[5]]
                $ 741 "write_welder(4, False )"
                write_welder(4,  False  )
              end
            end
            $ 742 "b2_par_cd≔0"
            global b2_par_cd=0
            $ 743 "homeing()"
            homeing()
          else:
            $ 744 "Else" "noBreak"
            $ 745 "homeing()"
            homeing()
          end
          $ 746 "HOR_R"
          $ 747 "If A_Prepos_l[A_HOR_R]≠p[0,0,0,0,0,0]"
          if (A_Prepos_l[A_HOR_R] != p[0,0,0,0,0,0]):
            $ 748 "b2_left_par≔ False "
            global b2_left_par=  False
            $ 749 "b8_wv_2f≔ True "
            global b8_wv_2f=  True
            $ 750 "b7_tilt_degree≔[0,0,0]"
            global b7_tilt_degree=[0,0,0]
            $ 751 "A_sel_v≔A_HOR_R"
            global A_sel_v=A_HOR_R
            $ 752 "wv_direction≔-1"
            global wv_direction=-1
            $ 753 "Call MoveandTouchFun_2f"
            MoveandTouchFun_2f()
            $ 755 "If b1_cell_info_R≟A or b1_cell_info_R≟C or b1_cell_info_R≟c"
            if (b1_cell_info_R == A  or  b1_cell_info_R == C  or  b1_cell_info_R == c):
              $ 756 "If A_Prepos_l[A_VR1]≟p[0,0,0,0,0,0]"
              if (A_Prepos_l[A_VR1] == p[0,0,0,0,0,0]):
                $ 758 "g_tp≔A_Prepos_l[A_HOR_R]"
                global g_tp=A_Prepos_l[A_HOR_R]
                $ 759 "Folder"
                $ 760 "g_cp≔get_actual_tcp_pose()"
                global g_cp= get_actual_tcp_pose ()
                $ 761 "g_cp≔pose_trans(g_cp, p[0,0,0,d2r(-12),d2r(5),0])"
                global g_cp= pose_trans (g_cp, p[0,0,0,d2r(-12),d2r(5),0])
                $ 762 "MoveL"
                $ 763 "g_cp" "breakAfter"
                movel(pose_trans(Base, g_cp), a=0.08, v=0.08)
                $ 766 "for_x_HOR_R≔contact_fun(A_Touch_p[A_HOR_R],[-1*wv_direction,0,0],10000,15,15,  False)"
                global for_x_HOR_R=contact_fun(A_Touch_p[A_HOR_R],[-1*wv_direction,0,0],10000,15,15,  False)
                $ 767 "direction(p[0,0,0,0,0,0],[0,1,0],20,120,160)"
                direction(p[0,0,0,0,0,0],[0,1,0],20,120,160)
                $ 768 "write_welder(4, False )"
                write_welder(4,  False  )
              else:
                $ 769 "Else" "noBreak"
                $ 770 "for_x_HOR_R≔p[0,0,0,0,0,0]"
                global for_x_HOR_R=p[0,0,0,0,0,0]
              end
            end
            $ 771 "wv_direction≔1"
            global wv_direction=1
            $ 772 "If point_dist(A_Prepos_l[A_HOR_R], A_Prepos_l[A_VR1])>0.032"
            if (point_dist(A_Prepos_l[A_HOR_R], A_Prepos_l[A_VR1])>0.032):
              $ 773 "homeing()"
              homeing()
            end
          end
          $ 774 "VR1"
          $ 775 "If A_Prepos_l[A_VR1]≠p[0,0,0,0,0,0]"
          if (A_Prepos_l[A_VR1] != p[0,0,0,0,0,0]):
            $ 776 "b2_left_par≔ False "
            global b2_left_par=  False
            $ 777 "b8_wv_2f≔ False "
            global b8_wv_2f=  False
            $ 778 "b7_tilt_degree≔basic_tilt_3f"
            global b7_tilt_degree=basic_tilt_3f
            $ 779 "A_sel_v≔A_VR1"
            global A_sel_v=A_VR1
            $ 780 "A_sel_v_end≔A_VR1_END"
            global A_sel_v_end=A_VR1_END
            $ 781 "b2_par_cd≔0"
            global b2_par_cd=0
            $ 782 "If b1_cell_info_R≟A or b1_cell_info_R≟C or b1_cell_info_R≟c"
            if (b1_cell_info_R == A  or  b1_cell_info_R == C  or  b1_cell_info_R == c):
              $ 783 "Scallup_check≔ True "
              global Scallup_check=  True
            else:
              $ 784 "Else" "noBreak"
              $ 785 "Scallup_check≔ False "
              global Scallup_check=  False
            end
            $ 786 "Call MoveandTouchFun_3f"
            MoveandTouchFun_3f()
            $ 787 "If b1_cell_info_R≟A or b1_cell_info_R≟C or b1_cell_info_R≟c"
            if (b1_cell_info_R == A  or  b1_cell_info_R == C  or  b1_cell_info_R == c):
              $ 788 "If A_Prepos_l[A_HOR_R]≟p[0,0,0,0,0,0]"
              if (A_Prepos_l[A_HOR_R] == p[0,0,0,0,0,0]):
                $ 789 "direction(p[0,0,0,0,0,0],[0,1,0],8,120,160)"
                direction(p[0,0,0,0,0,0],[0,1,0],8,120,160)
                $ 790 "AAgcp≔get_actual_tcp_pose()"
                global AAgcp= get_actual_tcp_pose ()
                $ 791 "AAgangle≔up_right"
                global AAgangle=p[.445203173045, -.406687378356, -.031125942276, 2.308490741423, -1.066468937023, 1.322151316133]
                $ 792 "AAgtp≔p[AAgcp[0],AAgcp[1],AAgcp[2],AAgangle[3],AAgangle[4],AAgangle[5]]"
                global AAgtp=p[AAgcp[0],AAgcp[1],AAgcp[2],AAgangle[3],AAgangle[4],AAgangle[5]]
                $ 793 "MoveL"
                $ 794 "AAgtp" "breakAfter"
                movel(pose_trans(Base, AAgtp), a=0.08, v=0.08)
                $ 796 "for_z_VR1≔contact_fun(p[0,0,0,0,0,0],[0,0,-1],10000,15,15,  False)"
                global for_z_VR1=contact_fun(p[0,0,0,0,0,0],[0,0,-1],10000,15,15,  False)
                $ 797 "direction(p[0,0,0,0,0,0],[0,0,1],20,120,160)"
                direction(p[0,0,0,0,0,0],[0,0,1],20,120,160)
                $ 798 "write_welder(4, False )"
                write_welder(4,  False  )
              else:
                $ 799 "Else" "noBreak"
                $ 800 "for_z_VR1≔p[0,0,0,0,0,0]"
                global for_z_VR1=p[0,0,0,0,0,0]
              end
            end
          end
          $ 801 "HOR_MR"
          $ 802 "If A_Prepos_l[A_HOR_MR]≠p[0,0,0,0,0,0]"
          if (A_Prepos_l[A_HOR_MR] != p[0,0,0,0,0,0]):
            $ 803 "INIT"
            $ 804 "b2_left_par≔ False "
            global b2_left_par=  False
            $ 805 "b8_wv_2f≔ True "
            global b8_wv_2f=  True
            $ 806 "b7_tilt_degree≔[0,0,0]"
            global b7_tilt_degree=[0,0,0]
            $ 807 "A_sel_v≔A_HOR_MR"
            global A_sel_v=A_HOR_MR
            $ 808 "If b1_cell_info_R≟C or b1_cell_info_R≟D"
            if (b1_cell_info_R == C  or  b1_cell_info_R == D):
              $ 809 "wv_direction≔-1"
              global wv_direction=-1
              $ 810 "Call MoveFun_cd"
              MoveFun_cd()
              $ 811 "for_cal_xy≔contact_fun(p[0,0,0,0,0,0],[1,0,0],20000,20,20)"
              global for_cal_xy=contact_fun(p[0,0,0,0,0,0],[1,0,0],20000,20,20)
              $ 812 "direction(p[0,0,0,0,0,0],[-1,0,0],15,120,160)"
              direction(p[0,0,0,0,0,0],[-1,0,0],15,120,160)
              $ 813 "direction(p[0,0,0,0,0,0],[0,1,0],60,120,160)"
              direction(p[0,0,0,0,0,0],[0,1,0],60,120,160)
              $ 814 "direction(p[0,0,0,0,0,0],[1,0,0],20,120,160)"
              direction(p[0,0,0,0,0,0],[1,0,0],20,120,160)
              $ 815 "for_cal_x_wel≔contact_fun(p[0,0,0,0,0,0],[0,-1,0],20000,20,20)"
              global for_cal_x_wel=contact_fun(p[0,0,0,0,0,0],[0,-1,0],20000,20,20)
              $ 816 "direction(p[0,0,0,0,0,0],[0,1,0],20,120,160)"
              direction(p[0,0,0,0,0,0],[0,1,0],20,120,160)
              $ 817 "for_cal_zr≔contact_fun(p[0,0,0,0,0,0],[0,0,-1],20000,20,20)"
              global for_cal_zr=contact_fun(p[0,0,0,0,0,0],[0,0,-1],20000,20,20)
              $ 818 "direction(p[0,0,0,0,0,0],[0,0,1],20,120,160)"
              direction(p[0,0,0,0,0,0],[0,0,1],20,120,160)
              $ 819 "If A_Prepos_l[A_VR2]≟p[0,0,0,0,0,0]"
              if (A_Prepos_l[A_VR2] == p[0,0,0,0,0,0]):
                $ 820 "for_cal_y_wel≔contact_fun(p[0,0,0,0,0,0],[1,0,0],20000,20,20)"
                global for_cal_y_wel=contact_fun(p[0,0,0,0,0,0],[1,0,0],20000,20,20)
                $ 821 "direction(p[0,0,0,0,0,0],[-1,0,0],8,120,160)"
                direction(p[0,0,0,0,0,0],[-1,0,0],8,120,160)
              end
              $ 822 "for_cal_rot≔A_Touch_p[A_HOR_R]"
              global for_cal_rot=A_Touch_p[A_HOR_R]
              $ 823 "A_Touch_p[A_sel_v]=p[for_cal_xy[0],for_cal_xy[1],for_cal_zr[2],for_cal_rot[3],for_cal_rot[4],for_cal_rot[5]]"
              A_Touch_p[A_sel_v]=p[for_cal_xy[0],for_cal_xy[1],for_cal_zr[2],for_cal_rot[3],for_cal_rot[4],for_cal_rot[5]]
              $ 824 "A_Touch_p[A_sel_v]=pose_trans(A_Touch_p[A_sel_v], p[-Touch_dis/1000,0,0,0,0,0])"
              A_Touch_p[A_sel_v]= pose_trans (A_Touch_p[A_sel_v], p[-Touch_dis/1000,0,0,0,0,0])
              $ 825 "write_welder(4, False )"
              write_welder(4,  False  )
            else:
              $ 826 "Else" "noBreak"
              $ 827 "wv_direction≔-1"
              global wv_direction=-1
              $ 828 "for_cal_rot≔A_Touch_p[A_HOR_R]"
              global for_cal_rot=A_Touch_p[A_HOR_R]
              $ 829 "Call MoveFun_cd"
              MoveFun_cd()
              $ 830 "for_cal_y_wel≔contact_fun(p[0,0,0,0,0,0],[1,0,0],20000,20,20)"
              global for_cal_y_wel=contact_fun(p[0,0,0,0,0,0],[1,0,0],20000,20,20)
              $ 831 "vr2_p1≔for_cal_y_wel"
              global vr2_p1=for_cal_y_wel
              $ 832 "for_cal_y_wel[2]=for_cal_rot[2]"
              for_cal_y_wel[2]=for_cal_rot[2]
              $ 833 "dir_x_cal≔get_feature_Line(for_cal_rot,for_cal_y_wel)"
              global dir_x_cal=get_feature_Line(for_cal_rot,for_cal_y_wel)
              $ 834 "vr2_p2≔feature_offset(vr2_p1,p[0,0.02,0,0,0,0],dir_x_cal)"
              global vr2_p2=feature_offset(vr2_p1,p[0,0.02,0,0,0,0],dir_x_cal)
              $ 835 "direction(p[0,0,0,0,0,0],[-1,0,0],40,120,160)"
              direction(p[0,0,0,0,0,0],[-1,0,0],40,120,160)
              $ 836 "direction(p[0,0,0,0,0,0],[0,1,0],80,120,160)"
              direction(p[0,0,0,0,0,0],[0,1,0],80,120,160)
              $ 837 "for_cal_y_wel≔contact_fun(p[0,0,0,0,0,0],[1,0,0],20000,20,20)"
              global for_cal_y_wel=contact_fun(p[0,0,0,0,0,0],[1,0,0],20000,20,20)
              $ 838 "direction(p[0,0,0,0,0,0],[-1,0,0],5,120,160)"
              direction(p[0,0,0,0,0,0],[-1,0,0],5,120,160)
              $ 839 "direction(p[0,0,0,0,0,0],[0,-1,0],50,120,160)"
              direction(p[0,0,0,0,0,0],[0,-1,0],50,120,160)
              $ 840 "direction(p[0,0,0,0,0,0],[1,0,0],7,120,160)"
              direction(p[0,0,0,0,0,0],[1,0,0],7,120,160)
              $ 841 "for_cal_x_wel≔contact_fun(p[0,0,0,0,0,0],[0,1,0],20000,20,20)"
              global for_cal_x_wel=contact_fun(p[0,0,0,0,0,0],[0,1,0],20000,20,20)
              $ 842 "vr2_p3≔for_cal_x_wel"
              global vr2_p3=for_cal_x_wel
              $ 843 "get_ml≔get_feature_pose(for_cal_x_wel,for_cal_rot)"
              global get_ml=get_feature_pose(for_cal_x_wel,for_cal_rot)
              $ 845 "A_Touch_p[A_sel_v]=feature_offset(for_cal_rot,p[0,-get_ml[0]+(-cd_offset+cd_extra_dis)/1000,0,0,0,0],dir_x_cal)"
              A_Touch_p[A_sel_v]=feature_offset(for_cal_rot,p[0,-get_ml[0]+(-cd_offset+cd_extra_dis)/1000,0,0,0,0],dir_x_cal)
              $ 846 "vr2_p4≔A_Touch_p[A_HOR_MR]"
              global vr2_p4=A_Touch_p[A_HOR_MR]
              $ 847 "direction(p[0,0,0,0,0,0],[0,-1,0],5,120,160)"
              direction(p[0,0,0,0,0,0],[0,-1,0],5,120,160)
              $ 848 "direction(p[0,0,0,0,0,0],[-1,0,0],20,120,160)"
              direction(p[0,0,0,0,0,0],[-1,0,0],20,120,160)
              $ 849 "write_welder(4, False )"
              write_welder(4,  False  )
            end
            $ 850 "wv_direction≔1"
            global wv_direction=1
          end
          $ 851 "VR2"
          $ 852 "If A_Prepos_l[A_VR2]≠p[0,0,0,0,0,0]"
          if (A_Prepos_l[A_VR2] != p[0,0,0,0,0,0]):
            $ 853 "Init"
            $ 854 "b2_left_par≔ False "
            global b2_left_par=  False
            $ 855 "b8_wv_2f≔ False "
            global b8_wv_2f=  False
            $ 856 "b7_tilt_degree≔basic_tilt_3f"
            global b7_tilt_degree=basic_tilt_3f
            $ 857 "A_sel_v≔A_VR2"
            global A_sel_v=A_VR2
            $ 858 "A_sel_v_end≔A_VR2_END"
            global A_sel_v_end=A_VR2_END
            $ 859 "b2_par_cd≔1"
            global b2_par_cd=1
            $ 860 "If b1_cell_info_R≟A or b1_cell_info_R≟C or b1_cell_info_R≟c"
            if (b1_cell_info_R == A  or  b1_cell_info_R == C  or  b1_cell_info_R == c):
              $ 861 "Scallup_check≔ True "
              global Scallup_check=  True
            else:
              $ 862 "Else" "noBreak"
              $ 863 "Scallup_check≔ False "
              global Scallup_check=  False
            end
            $ 864 "If b1_cell_info_R≟d or b1_cell_info_R≟c"
            if (b1_cell_info_R == d  or  b1_cell_info_R == c):
              $ 865 "If vr2_p1≟p[0,0,0,0,0,0]"
              if (vr2_p1 == p[0,0,0,0,0,0]):
                $ 866 "Call MoveFun_cd"
                MoveFun_cd()
                $ 867 "vr2_p1≔contact_fun(p[0,0,0,0,0,0],[1,0,0],20000,20,20)"
                global vr2_p1=contact_fun(p[0,0,0,0,0,0],[1,0,0],20000,20,20)
                $ 868 "direction(p[0,0,0,0,0,0],[-1,0,0],20,120,160)"
                direction(p[0,0,0,0,0,0],[-1,0,0],20,120,160)
                $ 869 "direction(p[0,0,0,0,0,0],[0,1,0],10,120,160)"
                direction(p[0,0,0,0,0,0],[0,1,0],10,120,160)
                $ 870 "vr2_p2≔contact_fun(p[0,0,0,0,0,0],[1,0,0],20000,20,20)"
                global vr2_p2=contact_fun(p[0,0,0,0,0,0],[1,0,0],20000,20,20)
                $ 871 "direction(p[0,0,0,0,0,0],[-1,0,0],14,120,160)"
                direction(p[0,0,0,0,0,0],[-1,0,0],14,120,160)
                $ 872 "vr2_p3≔contact_fun(p[0,0,0,0,0,0],[0,1,0],20000,20,20)"
                global vr2_p3=contact_fun(p[0,0,0,0,0,0],[0,1,0],20000,20,20)
                $ 873 "direction(p[0,0,0,0,0,0],[0,-1,0],30,120,160)"
                direction(p[0,0,0,0,0,0],[0,-1,0],30,120,160)
                $ 874 "direction(p[0,0,0,0,0,0],[-1,0,0],20,120,160)"
                direction(p[0,0,0,0,0,0],[-1,0,0],20,120,160)
                $ 875 "vr2_p4≔contact_fun(p[0,0,0,0,0,0],[0,0,-1],20000,20,20)"
                global vr2_p4=contact_fun(p[0,0,0,0,0,0],[0,0,-1],20000,20,20)
                $ 876 "direction(p[0,0,0,0,0,0],[0,0,1],40,120,160)"
                direction(p[0,0,0,0,0,0],[0,0,1],40,120,160)
                $ 877 "A_Touch_p[A_sel_v]=touch_xyz_get_middle(vr2_p1,vr2_p2,vr2_p3,vr2_p4)"
                A_Touch_p[A_sel_v]=touch_xyz_get_middle(vr2_p1,vr2_p2,vr2_p3,vr2_p4)
                $ 878 "var_4≔A_Touch_p[A_sel_v]"
                global var_4=A_Touch_p[A_sel_v]
                $ 879 "var_4≔pose_trans(var_4, p[a6_callar_vert/1000,0,0,0,0,0])"
                global var_4= pose_trans (var_4, p[a6_callar_vert/1000,0,0,0,0,0])
                $ 880 "var_5≔get_actual_tcp_pose()"
                global var_5= get_actual_tcp_pose ()
                $ 881 "var_5[2]=var_4[2]"
                var_5[2]=var_4[2]
                $ 882 "var_5≔pose_trans(var_5, p[0,0,0,0,d2r(10),0])"
                global var_5= pose_trans (var_5, p[0,0,0,0,d2r(10),0])
                $ 883 "MoveL"
                $ 884 "var_5" "breakAfter"
                movel(pose_trans(Base, var_5), a=0.1, v=0.1)
                $ 885 "vr2_p1_up≔contact_fun(p[0,0,0,0,0,0],[1,0,0],20000,20,20)"
                global vr2_p1_up=contact_fun(p[0,0,0,0,0,0],[1,0,0],20000,20,20)
                $ 886 "direction(p[0,0,0,0,0,0],[-1,0,0],20,120,160)"
                direction(p[0,0,0,0,0,0],[-1,0,0],20,120,160)
                $ 887 "direction(p[0,0,0,0,0,0],[0,1,0],10,120,160)"
                direction(p[0,0,0,0,0,0],[0,1,0],10,120,160)
                $ 888 "vr2_p2_up≔contact_fun(p[0,0,0,0,0,0],[1,0,0],20000,20,20)"
                global vr2_p2_up=contact_fun(p[0,0,0,0,0,0],[1,0,0],20000,20,20)
                $ 889 "direction(p[0,0,0,0,0,0],[-1,0,0],14,120,160)"
                direction(p[0,0,0,0,0,0],[-1,0,0],14,120,160)
                $ 890 "vr2_p3_up≔contact_fun(p[0,0,0,0,0,0],[0,1,0],20000,20,20)"
                global vr2_p3_up=contact_fun(p[0,0,0,0,0,0],[0,1,0],20000,20,20)
                $ 891 "direction(p[0,0,0,0,0,0],[0,-1,0],30,120,160)"
                direction(p[0,0,0,0,0,0],[0,-1,0],30,120,160)
                $ 892 "direction(p[0,0,0,0,0,0],[-1,0,0],20,120,160)"
                direction(p[0,0,0,0,0,0],[-1,0,0],20,120,160)
              end
              $ 893 "A_Touch_p[A_sel_v+9]=touch_4point(vr2_p1_up,vr2_p2_up,vr2_p3_up)"
